(* IEC 61131-3 sources: CodesysTest/alpha/export (part 2) *)

(* ---- ElectricPressureBarFB.st ---- *)
FUNCTION_BLOCK ElectricPressureBarFB IMPLEMENTS IComponentStatus
VAR_INPUT
    enable : BOOL;
END_VAR
VAR_IN_OUT

END_VAR
VAR_OUTPUT
END_VAR
VAR
    electricPressureBarMotor : FB_FestoMotor();
    delay: TON := (PT := T#1S);
    state : PRESSURE_BAR_STATES;
    enableElectricPressureBarONS : R_TRIG();

    _mode : DEVICE_MODES;    // Auto-SemiAuto-Manual
    _ready : BOOL;            // Ready to be controlled
    _amOpenJaw : BOOL;    // Auto Mode Open Jaw Command
    _amCloseJaw : BOOL;     // Auto Mode Close Jaw Command
END_VAR

//    Function Block: ElectricPressureBarFB
//    Description: This function block is the state machine for the electric pressure bar
//
//    Created by: Ben Hess
//    Created Date: Monday, April 16, 2018

electricPressureBarMotor(deviceType := FML.CMMP_AS,
                                        isFPCActive := TRUE,
                                        ptrReadFHPPRegister := ADR(%IW145),
                                        ptrReadFPCRegister := ADR(%IW149),
                                        ptrWriteFHPPRegister := ADR(%QW82),
                                        ptrWriteFPCRegister := ADR(%QW86));
electricPressureBarMotor.Execute();

delay();

//Report as ready if mode is auto and we're not faulted
_ready := (_mode = DEVICE_MODES.Auto) AND NOT (state = PRESSURE_BAR_STATES.Fault);

enableElectricPressureBarONS(CLK := enable);
IF enableElectricPressureBarONS.Q THEN
    state := PRESSURE_BAR_STATES.Idle;
END_IF

IF NOT enable THEN
        state := PRESSURE_BAR_STATES.Fault;
END_IF

CASE state OF
    PRESSURE_BAR_STATES.Idle:        IF enable AND _mode = DEVICE_MODES.SemiAuto OR (_mode = DEVICE_MODES.Auto AND _amCloseJaw) THEN
                                        state := PRESSURE_BAR_STATES.CloseJaw;
                                        _amCloseJaw := FALSE;
                                    END_IF

    PRESSURE_BAR_STATES.OpenJaw:    electricPressureBarMotor.ExecuteStoredProgram(1);
                                    IF electricPressureBarMotor.CommandAcknowledged THEN
                                        state := PRESSURE_BAR_STATES.OpeningJaw;
                                        Globals.electricPressureBarCount := Globals.electricPressureBarCount + 1;
                                    END_IF

    PRESSURE_BAR_STATES.OpeningJaw:
                                    IF electricPressureBarMotor.ActiveStoredProgramNumber = 1 AND electricPressureBarMotor.InPosition THEN
                                        state := PRESSURE_BAR_STATES.JawOpened;
                                    END_IF

    PRESSURE_BAR_STATES.JawOpened:     IF _mode = DEVICE_MODES.SemiAuto THEN
                                        delay.IN := TRUE;
                                        IF delay.Q THEN
                                            state := PRESSURE_BAR_STATES.CloseJaw;
                                            delay.IN := FALSE;
                                        END_IF
                                    ELSIF _mode = DEVICE_MODES.Auto AND _amCloseJaw THEN
                                        state := PRESSURE_BAR_STATES.CloseJaw;
                                        _amCloseJaw := FALSE;
                                    END_IF

    PRESSURE_BAR_STATES.CloseJaw:    electricPressureBarMotor.ExecuteStoredProgram(2);
                                    IF electricPressureBarMotor.CommandAcknowledged THEN
                                        state := PRESSURE_BAR_STATES.ClosingJaw;
                                        Globals.electricPressureBarCount := Globals.electricPressureBarCount + 1;
                                    END_IF

    PRESSURE_BAR_STATES.ClosingJaw:    IF electricPressureBarMotor.ActiveStoredProgramNumber = 2 AND electricPressureBarMotor.InPosition THEN
                                        state := PRESSURE_BAR_STATES.JawClosed;
                                    END_IF

    PRESSURE_BAR_STATES.JawClosed:    IF _mode = DEVICE_MODES.SemiAuto THEN
                                        delay.IN := TRUE;
                                        IF delay.Q THEN
                                            state := PRESSURE_BAR_STATES.OpenJaw;
                                            delay.IN := FALSE;
                                        END_IF
                                    ELSIF _mode = DEVICE_MODES.Auto AND _amOpenJaw THEN
                                        state := PRESSURE_BAR_STATES.OpenJaw;
                                        _amOpenJaw := FALSE;
                                    END_IF

    PRESSURE_BAR_STATES.Fault:        ClearCommands();

END_CASE

METHOD AutoCloseJaw
VAR_INPUT
END_VAR

_amCloseJaw := TRUE;

METHOD AutoOpenJaw
VAR_INPUT
END_VAR

_amOpenJaw := TRUE;

PROPERTY Mode : DEVICE_MODES

PROPERTY Ready : BOOL

METHOD PRIVATE ClearCommands
VAR_INPUT
END_VAR

_amCloseJaw := FALSE;
_amOpenJaw := FALSE;

(* ---- FB_AppliedMotionBagDeliveryMotor.st ---- *)
FUNCTION_BLOCK FB_AppliedMotionBagDeliveryMotor EXTENDS FB_AppliedMotionStepServoTCP
VAR_INPUT
END_VAR
VAR_OUTPUT
END_VAR
VAR
    sendParameters : FB_SendUserRegistersAppliedMotionTCP();
    sendBagMoveCommand : FB_SendBagMoveAppliedMotionTCP();
END_VAR

sendMoveCommand(Slave := slave);
sendBagMoveCommand(Slave := slave);
sendOpcodeCommand(Slave := slave);
sendParameters(Slave := slave);

commandSuccessful S= ((sendMoveCommand.xDone OR sendOpcodeCommand.xDone OR sendBagMoveCommand.xDone) AND NOT status.inPosition) OR sendParameters.xDone;

METHOD MoveDistance
VAR_INPUT
    distance : REAL;        //Distance to move in inches
    acceleration : INT;        //Acceleration in RPM/sec
    deceleration : INT;        //Deceleration in RPM/sec
    velocity : INT;            //Velocity in .25RPM
END_VAR
distanceToMoveInSteps.rawValue := REAL_TO_DINT((distance) * stepsPerInchSetpoint);
IF reversePolarity THEN
    distanceToMoveInSteps.rawValue := distanceToMoveInSteps.rawValue * -1;
END_IF
commandSuccessful := FALSE;
ModbusLongHandler.Unpack(distanceToMoveInSteps);
sendBagMoveCommand.acceleration := acceleration;
sendBagMoveCommand.deceleration := deceleration;
sendBagMoveCommand.velocity := velocity;
sendBagMoveCommand.distanceHighWord := distanceToMoveInSteps.highWord;
sendBagMoveCommand.distanceLowWord := distanceToMoveInSteps.lowWord;
sendBagMoveCommand.opcode := STEP_SERVO_OPCODES.QUEUE_LOAD_AND_EXECUTE;
sendBagMoveCommand.programToRun := 1;
sendBagMoveCommand.Execute();

METHOD SendParameters
VAR_INPUT
    reverseSpeed : DINT;

END_VAR

METHOD MoveDistanceFinal
VAR_INPUT
    distance : REAL;        //Distance to move in inches
    acceleration : INT;        //Acceleration in RPM/sec
    deceleration : INT;        //Deceleration in RPM/sec
    velocity : INT;            //Velocity in .25RPM
END_VAR

distanceToMoveInSteps.rawValue := REAL_TO_DINT((distance) * stepsPerInchSetpoint);
IF reversePolarity THEN
    distanceToMoveInSteps.rawValue := distanceToMoveInSteps.rawValue * -1;
END_IF
commandSuccessful := FALSE;
ModbusLongHandler.Unpack(distanceToMoveInSteps);
sendBagMoveCommand.acceleration := acceleration;
sendBagMoveCommand.deceleration := deceleration;
sendBagMoveCommand.velocity := velocity;
sendBagMoveCommand.distanceHighWord := distanceToMoveInSteps.highWord;
sendBagMoveCommand.distanceLowWord := distanceToMoveInSteps.lowWord;
sendBagMoveCommand.opcode := STEP_SERVO_OPCODES.QUEUE_LOAD_AND_EXECUTE;
sendBagMoveCommand.programToRun := 2;
sendBagMoveCommand.Execute();

METHOD StopViaProgram

// Load program segment 12 into buffer and execute.  This program contains nothing but a SM command.
// We must do it this way because the normal "stop command" opcode we have access to over modbus
// also kills the program buffer which is bad.
commandSuccessful := FALSE;
SendOpcodeCommand.opcode := STEP_SERVO_OPCODES.QUEUE_LOAD_AND_EXECUTE;
SendOpcodeCommand.Parameter1 := INT_TO_WORD(12);    //program 12 is just a SM command
SendOpcodeCommand.Execute();

(* ---- FB_AppliedMotionBagDeliveryMotor_1.st ---- *)
FUNCTION_BLOCK FB_AppliedMotionBagDeliveryMotor_1 EXTENDS FB_AppliedMotionStepServoEIPBase
VAR_INPUT
END_VAR
VAR_OUTPUT
END_VAR
VAR
	_moveDistance : BOOL;
	_moveDistanceONS : R_TRIG;
	_moveFinal : BOOL;
	_moveFinalONS : R_TRIG;
	_moveDone : BOOL;
	waitForMove : TON := (PT := T#30MS);
	manualFinalMovePB : BOOL;
	movedFinal : BOOL;
	moveDistanceState : AMP_EIP_MOVE_INITIAL_STATES;
	moveDistanceFinalState : AMP_EIP_MOVE_INITIAL_STATES;
END_VAR

METHOD Execute
VAR_INPUT
END_VAR

SUPER^.Execute();
waitForMove();
_moveDistanceONS(CLK := _moveDistance);
_moveFinalONS(CLK := _moveFinal);

CASE moveDistanceState OF
	AMP_EIP_MOVE_INITIAL_STATES.Idle :
															IF _moveDistance THEN
																moveDistanceState := AMP_EIP_MOVE_INITIAL_STATES.SetOutputOff;
															END_IF

	AMP_EIP_MOVE_INITIAL_STATES.SetOutputOff :					sclCommand := 16#534F; //Output off
															parameter1 := 16#48B2;
															commands.SendHostCommand := TRUE;
															IF commandSuccessful THEN
																commandSuccessful := FALSE;
																moveDistanceState := AMP_EIP_MOVE_INITIAL_STATES.WaitAfterSettingOutputOff;
															END_IF

	AMP_EIP_MOVE_INITIAL_STATES.WaitAfterSettingOutputOff :
															IF commandSuccessful THEN
																moveDistanceState := AMP_EIP_MOVE_INITIAL_STATES.MoveMotor;
															END_IF

	AMP_EIP_MOVE_INITIAL_STATES.MoveMotor: 					commandSuccessful := FALSE;
															sclCommand := 16#0;
															parameter1 := 16#0;
															commands.FeedToLength := TRUE;
															_moveDistance := FALSE;
															moveDistanceState := AMP_EIP_MOVE_INITIAL_STATES.WaitAfterMovingMotor;

	AMP_EIP_MOVE_INITIAL_STATES.WaitAfterMovingMotor: 		IF commandSuccessful THEN
																_moveDone := TRUE;
																moveDistanceState := AMP_EIP_MOVE_INITIAL_STATES.Idle;
															END_IF
END_CASE

CASE moveDistanceFinalState OF
	AMP_EIP_MOVE_INITIAL_STATES.Idle :						IF _moveFinal THEN
																moveDistanceFinalState := AMP_EIP_MOVE_INITIAL_STATES.SetOutputOff;
															END_IF

	AMP_EIP_MOVE_INITIAL_STATES.SetOutputOff :					sclCommand := 16#534F; //Output off
															parameter1 := 16#48B2;
															commands.SendHostCommand := TRUE;
															IF commandSuccessful THEN
																commandSuccessful := FALSE;
																moveDistanceFinalState := AMP_EIP_MOVE_INITIAL_STATES.WaitAfterSettingOutputOff;
															END_IF

	AMP_EIP_MOVE_INITIAL_STATES.WaitAfterSettingOutputOff :
															IF commandSuccessful THEN
																moveDistanceFinalState := AMP_EIP_MOVE_INITIAL_STATES.MoveMotor;
															END_IF

	AMP_EIP_MOVE_INITIAL_STATES.MoveMotor: 					sclCommand := 16#0;
															parameter1 := 16#0;
															commandSuccessful := FALSE;
															commands.FeedToLength := TRUE;
															moveDistanceFinalState := AMP_EIP_MOVE_INITIAL_STATES.WaitAfterMovingMotor;

	AMP_EIP_MOVE_INITIAL_STATES.WaitAfterMovingMotor: 		IF commandSuccessful AND InPosition THEN
																moveDistanceFinalState := AMP_EIP_MOVE_INITIAL_STATES.SetOutputOn;
															END_IF

	AMP_EIP_MOVE_INITIAL_STATES.SetOutputOn :					sclCommand := 16#534F; // Output on
															parameter1 := 16#4CB2;

															commandSuccessful := FALSE;
															commands.SendHostCommand := TRUE;
															_moveFinal := FALSE;
															moveDistanceFinalState := AMP_EIP_MOVE_INITIAL_STATES.WaitAfterSettingOutputOn;

	AMP_EIP_MOVE_INITIAL_STATES.WaitAfterSettingOutputOn :
															IF commandSuccessful THEN
																_moveDone := TRUE;
																moveDistanceFinalState := AMP_EIP_MOVE_INITIAL_STATES.Idle;
															END_IF

END_CASE
(*
IF _moveFinal THEN
	IF NOT movedFinal AND commandSuccessful THEN
		commandSuccessful := FALSE;
		commands.FeedToLength := TRUE;
		waitForMove.IN := TRUE;
		movedFinal := TRUE;
	END_IF

	IF commandSuccessful AND waitForMove.Q AND InPosition THEN
		sclCommand := 16#534F;
		parameter1 := 16#4CB2;
		commands.SendHostCommand := TRUE;
		_moveFinal := FALSE;
		waitForMove.IN := FALSE;
		movedFinal := FALSE;
	END_IF
END_IF
*)
IF manualFinalMovePB THEN
    MoveDistanceFinal(distance := distanceSetpointInches, acceleration := pointToPointAccelSetpoint, deceleration := pointToPointDecelSetpoint, velocity := velocitySetpoint);
    manualFinalMovePB := FALSE;
END_IF

PROPERTY CommandAcknowledged : BOOL

METHOD SetRearMotorToTorqueMode
VAR_INPUT
END_VAR

sclCommand := 16#534F; // Output on
parameter1 := 16#4CB2;

commandSuccessful := FALSE;
commands.SendHostCommand := TRUE;

METHOD SetRearMotorToEncoderFollowing
VAR_INPUT
END_VAR

METHOD StopViaProgram

// Load program segment 12 into buffer and execute.  This program contains nothing but a SM command.
// We must do it this way because the normal "stop command" opcode we have access to over modbus
// also kills the program buffer which is bad.
SUPER^.Stop();

METHOD MoveDistanceFinal
VAR_INPUT
    distance : REAL;        //Distance to move in inches
    acceleration : INT;        //Acceleration in RPM/sec
    deceleration : INT;        //Deceleration in RPM/sec
    velocity : INT;            //Velocity in .25RPM
END_VAR

commandSuccessful := FALSE;
_moveDone := FALSE;
moveDistanceFinalState := AMP_EIP_MOVE_INITIAL_STATES.Idle;
distanceToMoveInSteps := REAL_TO_DINT((distance) * stepsPerInchSetpoint);
IF reversePolarity THEN
    distanceToMoveInSteps := distanceToMoveInSteps * -1;
END_IF

pointToPointAccelSetpoint := acceleration;
pointToPointDecelSetpoint := deceleration;
velocitySetpoint := velocity;

currentLimit := defaultCurrentSetpoint;
_moveFinal := TRUE;
//SUPER^.ExecuteStoredProgram(2);

METHOD MoveDistance
VAR_INPUT
    distance : REAL;        //Distance to move in inches
    acceleration : INT;        //Acceleration in RPM/sec
    deceleration : INT;        //Deceleration in RPM/sec
    velocity : INT;            //Velocity in .25RPM
END_VAR
commandSuccessful := FALSE;
_moveDone := FALSE;
moveDistanceState := AMP_EIP_MOVE_INITIAL_STATES.Idle;
distanceToMoveInSteps := REAL_TO_DINT((distance) * stepsPerInchSetpoint);

IF reversePolarity THEN
    distanceToMoveInSteps := distanceToMoveInSteps * -1;
END_IF

pointToPointAccelSetpoint := acceleration;
pointToPointDecelSetpoint := deceleration;
velocitySetpoint := velocity;

currentLimit := defaultCurrentSetpoint;
_moveDistance := TRUE;

//commands.feedToLength := TRUE;
//SUPER^.ExecuteStoredProgram(1);

(* ---- FB_AppliedMotionBagDeliveryMotorNoFollowing.st ---- *)
FUNCTION_BLOCK FB_AppliedMotionBagDeliveryMotorNoFollowing EXTENDS FB_AppliedMotionStepServoEIPBase
VAR_INPUT
END_VAR
VAR_OUTPUT
END_VAR
VAR
	_moveDistance : BOOL;
	_moveDistanceONS : R_TRIG;
	_moveFinal : BOOL;
	_moveFinalONS : R_TRIG;
	_moveDone : BOOL;
	waitForMove : TON := (PT := T#30MS);
	manualFinalMovePB : BOOL;
	movedFinal : BOOL;
	moveDistanceState : AMP_EIP_MOVE_INITIAL_STATES;
	moveDistanceFinalState : AMP_EIP_MOVE_INITIAL_STATES;
END_VAR

METHOD Execute
VAR_INPUT
END_VAR

SUPER^.Execute();
waitForMove();
_moveDistanceONS(CLK := _moveDistance);
_moveFinalONS(CLK := _moveFinal);

CASE moveDistanceState OF
	AMP_EIP_MOVE_INITIAL_STATES.Idle :
															IF _moveDistance THEN
																moveDistanceState := AMP_EIP_MOVE_INITIAL_STATES.SetOutputOff;
															END_IF

	AMP_EIP_MOVE_INITIAL_STATES.SetOutputOff :					sclCommand := 16#534F; //Output off
															parameter1 := 16#48B2;
															commands.SendHostCommand := TRUE;
															IF commandSuccessful THEN
																commandSuccessful := FALSE;
																moveDistanceState := AMP_EIP_MOVE_INITIAL_STATES.WaitAfterSettingOutputOff;
															END_IF

	AMP_EIP_MOVE_INITIAL_STATES.WaitAfterSettingOutputOff :
															IF commandSuccessful THEN
																moveDistanceState := AMP_EIP_MOVE_INITIAL_STATES.MoveMotor;
															END_IF

	AMP_EIP_MOVE_INITIAL_STATES.MoveMotor: 					commandSuccessful := FALSE;
															sclCommand := 16#0;
															parameter1 := 16#0;
															commands.FeedToLength := TRUE;
															_moveDistance := FALSE;
															moveDistanceState := AMP_EIP_MOVE_INITIAL_STATES.WaitAfterMovingMotor;

	AMP_EIP_MOVE_INITIAL_STATES.WaitAfterMovingMotor: 		IF commandSuccessful THEN
																_moveDone := TRUE;
																moveDistanceState := AMP_EIP_MOVE_INITIAL_STATES.Idle;
															END_IF
END_CASE

CASE moveDistanceFinalState OF
	AMP_EIP_MOVE_INITIAL_STATES.Idle :						IF _moveFinal THEN
																moveDistanceFinalState := AMP_EIP_MOVE_INITIAL_STATES.MoveMotor;
															END_IF

	AMP_EIP_MOVE_INITIAL_STATES.MoveMotor: 					sclCommand := 16#0;
															parameter1 := 16#0;
															commandSuccessful := FALSE;
															commands.FeedToLength := TRUE;
															moveDistanceFinalState := AMP_EIP_MOVE_INITIAL_STATES.WaitAfterMovingMotor;

	AMP_EIP_MOVE_INITIAL_STATES.WaitAfterMovingMotor: 		IF commandSuccessful AND InPosition THEN
																moveDistanceFinalState := AMP_EIP_MOVE_INITIAL_STATES.SetOutputOff;
															END_IF

	AMP_EIP_MOVE_INITIAL_STATES.SetOutputOff :					sclCommand := 16#534F; // Output on
															parameter1 := 16#4CB2;

															commandSuccessful := FALSE;
															commands.SendHostCommand := TRUE;
															_moveFinal := FALSE;
															moveDistanceFinalState := AMP_EIP_MOVE_INITIAL_STATES.WaitAfterSettingOutputOff;

	AMP_EIP_MOVE_INITIAL_STATES.WaitAfterSettingOutputOff :
															IF commandSuccessful THEN
																_moveDone := TRUE;
																moveDistanceFinalState := AMP_EIP_MOVE_INITIAL_STATES.Idle;
															END_IF

END_CASE
(*
IF _moveFinal THEN
	IF NOT movedFinal AND commandSuccessful THEN
		commandSuccessful := FALSE;
		commands.FeedToLength := TRUE;
		waitForMove.IN := TRUE;
		movedFinal := TRUE;
	END_IF

	IF commandSuccessful AND waitForMove.Q AND InPosition THEN
		sclCommand := 16#534F;
		parameter1 := 16#4CB2;
		commands.SendHostCommand := TRUE;
		_moveFinal := FALSE;
		waitForMove.IN := FALSE;
		movedFinal := FALSE;
	END_IF
END_IF
*)
IF manualFinalMovePB THEN
    MoveDistanceFinal(distance := distanceSetpointInches, acceleration := pointToPointAccelSetpoint, deceleration := pointToPointDecelSetpoint, velocity := velocitySetpoint);
    manualFinalMovePB := FALSE;
END_IF

PROPERTY CommandAcknowledged : BOOL

METHOD SetRearMotorToTorqueMode
VAR_INPUT
END_VAR

METHOD SetRearMotorToEncoderFollowing
VAR_INPUT
END_VAR

METHOD StopViaProgram

// Load program segment 12 into buffer and execute.  This program contains nothing but a SM command.
// We must do it this way because the normal "stop command" opcode we have access to over modbus
// also kills the program buffer which is bad.
SUPER^.Stop();

METHOD MoveDistanceFinal
VAR_INPUT
    distance : REAL;        //Distance to move in inches
    acceleration : INT;        //Acceleration in RPM/sec
    deceleration : INT;        //Deceleration in RPM/sec
    velocity : INT;            //Velocity in .25RPM
END_VAR

commandSuccessful := FALSE;
_moveDone := FALSE;
moveDistanceFinalState := AMP_EIP_MOVE_INITIAL_STATES.Idle;
distanceToMoveInSteps := REAL_TO_DINT((distance) * stepsPerInchSetpoint);
IF reversePolarity THEN
    distanceToMoveInSteps := distanceToMoveInSteps * -1;
END_IF

pointToPointAccelSetpoint := acceleration;
pointToPointDecelSetpoint := deceleration;
velocitySetpoint := velocity;

currentLimit := defaultCurrentSetpoint;
_moveFinal := TRUE;
//SUPER^.ExecuteStoredProgram(2);

METHOD MoveDistance
VAR_INPUT
    distance : REAL;        //Distance to move in inches
    acceleration : INT;        //Acceleration in RPM/sec
    deceleration : INT;        //Deceleration in RPM/sec
    velocity : INT;            //Velocity in .25RPM
END_VAR
commandSuccessful := FALSE;
_moveDone := FALSE;
moveDistanceState := AMP_EIP_MOVE_INITIAL_STATES.Idle;
distanceToMoveInSteps := REAL_TO_DINT((distance) * stepsPerInchSetpoint);

IF reversePolarity THEN
    distanceToMoveInSteps := distanceToMoveInSteps * -1;
END_IF

pointToPointAccelSetpoint := acceleration;
pointToPointDecelSetpoint := deceleration;
velocitySetpoint := velocity;

currentLimit := defaultCurrentSetpoint;
_moveDistance := TRUE;

//commands.feedToLength := TRUE;
//SUPER^.ExecuteStoredProgram(1);

(* ---- FB_AppliedMotionStepServoEIPBase.st ---- *)
FUNCTION_BLOCK FB_AppliedMotionStepServoEIPBase IMPLEMENTS IPositionableMotor, IStoredProgramMotor
VAR_INPUT
    ptrEIPInputs : POINTER TO ARRAY[0..13] OF  DINT;
    ptrEIPOutputs : POINTER TO ARRAY[0..15] OF DINT;
    faultHandler : REFERENCE TO FB_FaultHandler;
	commFail : BOOL;
    stepsPerInchSetpoint : INT;             //Steps per inch setpoint
    reversePolarity : BOOL;                 //0 = Normal, 1 = reversed polarity for display
    jogAccelSetpoint : INT;        //Point-to-Point Acceleration (AC) Setpoint
    jogDecelSetpoint : INT;        //Point-to-Point Deceleration (DE) Setpoint
    jogVelocitySetpoint : INT;                //Velocity (VE) Setpoint
    pointToPointAccelSetpoint : INT;        //Point-to-Point Acceleration (AC) Setpoint
    pointToPointDecelSetpoint : INT;        //Point-to-Point Deceleration (DE) Setpoint
    velocitySetpoint : INT;                //Velocity (VE) Setpoint
	defaultCurrentSetpoint : DINT;
	sclCommand : DINT;						// SCL Command from
	parameter1 : DINT;						// Data/SCL parameter 1
	parameter2 : DINT;						// Data/SCL parameter 2
    distanceSetpointInches : REAL;        //Distance setpoint in inches Setpoint
    moveDistanceManualPB : BOOL;            //Move distance pushbutton
    movePositionManualPB : BOOL;            //Move position pushbutton
	isHomable : BOOL;
END_VAR
VAR_IN_OUT
    //slave : IoDrvModbusTCP.ModbusTCPSlave;                    //Slave ModbusTCP Object
END_VAR
VAR
    absolutePositionSteps : DINT; //Immediate Absolute Position in steps
    distanceToMoveInSteps : DINT;        //Distance Setpoint to Drive
    stepServoStatusRaw : INT; //Raw step servo status over modbus
	stepServoAlarmCodeRaw : INT; // Ras Step Servo alarm code word
	currentLimit : DINT;
    commands : FB_StepServoCommands();
    commandSuccessful : BOOL;    //Modbus Command was successful
    commandSuccessfulONS : R_TRIG;    //Modbus Command was successful
    commandSentONS : R_TRIG;    //Modbus Command was successful
    homeRequiredIndication : BOOL; //Home required indication.
    driveInputs : ARRAY[0..13] OF DINT;        // Inputs from drive over EIP
    driveOutputs : ARRAY[0..15] OF DINT;    // Outputs to drive over EIP
    interfaceToPass : IFault;
    faultListRegisterSuccess : BOOL;        // Registering in fault list successful
    _faulted : BOOL;                    // Motor Faulted
	_reset : BOOL;			//Reset Motor
	_homeNow : BOOL;
	homingOSF : F_TRIG;

	IECReferenceGood : BOOL;
END_VAR
VAR_OUTPUT
    absolutePositonInches : REAL; //Immediate Absolute Positon in inches
    velocity : INT;    //Velocity (VE) Input from Drive
    status : StepServoStatusFB; //Status of servo
	alarms : FB_StepServoAlarms; // Alarms from Drive
    QSegmentRunning : INT; //Current Q program running from Drive
	faults : StepServoFaultsType;
END_VAR

IF NOT faultListRegisterSuccess THEN
    faultListRegisterSuccess := RegisterWithFaultHandler();
END_IF

{attribute 'monitoring' := 'variable'}
PROPERTY HomeRequired : BOOL

{attribute 'monitoring' := 'variable'}
PROPERTY InPosition : BOOL

//{warning 'add method implementation '}
METHOD Stop

commandSuccessful := FALSE;
commands.StopNormal := TRUE;

METHOD RegisterWithFaultHandler : BOOL

// If faulthandler hasn't been initialized yet then do nothing.

(*
IF NOT __ISVALIDREF(faultHandler) THEN
     RETURN;
END_IF

interfaceToPass := THIS^;
faultHandler.registerFaultSource(interfaceToPass);
RegisterWithFaultHandler := TRUE;
*)

{attribute 'monitoring' := 'variable'}
PROPERTY Faulted : BOOL

{attribute 'monitoring' := 'variable'}
PROPERTY Homing : BOOL

METHOD Execute
VAR_INPUT
END_VAR

//    Function Block: AppliedMotionStepServo
//    Description: This block provides an abstraction for a Ethernet I/P Applied Motion Step Servo
//    Created by: Ben Hess
//    Created Date: May 11th, 2018

// Use pointers for EIP memory register locations
driveInputs := ptrEIPInputs^;
// Step servo command bits handler
commands();
ptrEIPOutputs^ := driveOutputs;
alarms(alarmCode := stepServoAlarmCodeRaw, faults := faults);

IF currentLimit = 0 THEN
	currentLimit := defaultCurrentSetpoint;
END_IF
//Map raw EIP Registers to parameters
absolutePositionSteps := driveInputs[6];
velocity := DINT_TO_INT(driveInputs[8]);
stepServoStatusRaw := DINT_TO_INT(driveInputs[0]);

driveOutputs[4] := velocitySetpoint;
driveOutputs[5] := pointToPointAccelSetpoint;
driveOutputs[6] := pointToPointDecelSetpoint;
driveOutputs[7] := distanceToMoveInSteps;
driveOutputs[8] := currentLimit;
driveOutputs[9] := sclCommand;
driveOutputs[10] := parameter1;
driveOutputs[11] := parameter2;
driveOutputs[12] := currentLimit;
driveOutputs[13] := currentLimit + 1;
driveOutputs[0] := commands.commandWord;

//Convert Distance setpoint to steps.  Reverse polarity for display purposes if needed.

absolutePositonInches := (DINT_TO_REAL(absolutePositionSteps) / INT_TO_REAL(stepsPerInchSetpoint));

//Homing required from motor - for now just if there was an initialization seen.
homeRequiredIndication S= status.initializing OR Globals.firstScan OR _faulted OR driveInputs[11].0;

homingOSF(CLK := status.homing);
IF NOT driveInputs[11].0 THEN
	homeRequiredIndication := FALSE;
END_IF

commandSentONS(CLK := commands.commandSent);

IF commandSentONS.Q THEN
	commandSuccessful := TRUE;
END_IF

commandSuccessfulONS(CLK := commandSuccessful);
IF commandSuccessfulONS.Q THEN
	//parameter1 := 0;
	//velocitySetpoint := 0;
	//pointToPointAccelSetpoint := 0;
	//pointToPointDecelSetpoint := 0;
	//distanceToMoveInSteps := 0;
END_IF

IF _reset AND (status.driveFaulted OR status.alarmPresent) THEN
	commands.alarmReset := TRUE;
	_reset := FALSE;
END_IF

IF reversePolarity THEN
    absolutePositonInches := absolutePositonInches * -1;
END_IF

//Get Servo Status and unpack
status(statusCode := StepServoStatusRaw);

//Bit-packing for LONG types over Modbus

_faulted := status.driveFaulted OR status.alarmPresent OR commFail;

//Manual moves for motor
IF moveDistanceManualPB THEN
    MoveDistance(distance := distanceSetpointInches, acceleration := pointToPointAccelSetpoint, deceleration := pointToPointDecelSetpoint, velocity := velocitySetpoint);
    moveDistanceManualPB := FALSE;
END_IF

IF movePositionManualPB THEN
    MoveToPosition(position := distanceSetpointInches, acceleration := pointToPointAccelSetpoint, deceleration := pointToPointDecelSetpoint, velocity := velocitySetpoint);
    movePositionManualPB := FALSE;
END_IF

faults.commFail.faultTrigger := commFail AND Globals.machinePowerOK;
faults.notHomed.faultTrigger := homeRequiredIndication AND isHomable;

METHOD MoveDistance
VAR_INPUT
    (*Distance to move in inches*)
    distance    : REAL;
    (*Acceleration in RPM/sec*)
    acceleration    : INT;
    (*Deceleration in RPM/sec*)
    deceleration    : INT;
    (*Velocity in .25RPM*)
    velocity    : INT;
END_VAR

//This method preps the data to send to the drive and triggers the send.
//Set distance and unpack to prep data to send to motor

commandSuccessful := FALSE;

distanceToMoveInSteps := REAL_TO_DINT((distance) * stepsPerInchSetpoint);
IF reversePolarity THEN
    distanceToMoveInSteps := distanceToMoveInSteps * -1;
END_IF

pointToPointAccelSetpoint := acceleration;
pointToPointDecelSetpoint := deceleration;
velocitySetpoint := velocity;
currentLimit := defaultCurrentSetpoint;

commands.feedToLength := TRUE;

METHOD HomeNow
commandSuccessful := FALSE;
parameter1 := 1;
pointToPointAccelSetpoint := 1000;
pointToPointDecelSetpoint := 1000;
velocitySetpoint := 2500;
distanceToMoveInSteps := 0;
commands.sendQAndExecute := TRUE;

//homeRequiredIndication := FALSE;

{attribute 'monitoring' := 'variable'}
PROPERTY CurrentPosition : REAL  //Current motor position in Inches

METHOD ExecuteStoredProgram
VAR_INPUT
    (*Program number to execute*)
    programNumber    : INT;
END_VAR

parameter1 := programNumber;
commands.SendQAndExecute := TRUE;

{attribute 'monitoring' := 'variable'}
PROPERTY Moving : BOOL

{attribute 'monitoring' := 'variable'}
PROPERTY ActiveStoredProgramNumber : INT

METHOD MoveDistanceTorque
VAR_INPUT
	(*Distance to move in inches*)
    distance    : REAL;
    (*Acceleration in RPM/sec*)
    acceleration    : INT;
    (*Deceleration in RPM/sec*)
    deceleration    : INT;
    (*Velocity in .25RPM*)
    velocity    : INT;
	(*Current in .01A*)
	current : DINT;
END_VAR

//This method preps the data to send to the drive and triggers the send.
//Set distance and unpack to prep data to send to motor

commandSuccessful := FALSE;

distanceToMoveInSteps := REAL_TO_DINT((distance) * stepsPerInchSetpoint);
IF reversePolarity THEN
    distanceToMoveInSteps := distanceToMoveInSteps * -1;
END_IF

pointToPointAccelSetpoint := acceleration;
pointToPointDecelSetpoint := deceleration;
velocitySetpoint := velocity;
currentLimit := current;

commands.feedToLength := TRUE;

METHOD Reset : BOOL
VAR_INPUT
END_VAR

IF Faulted THEN
	_reset := TRUE;
	commands.AlarmReset := TRUE;
END_IF
commands.Enable := TRUE;

{attribute 'monitoring' := 'variable'}
PROPERTY CommandAcknowledged : BOOL

(* ---- FB_AppliedMotionStepServoEIPBaseQX.st ---- *)
FUNCTION_BLOCK FB_AppliedMotionStepServoEIPBaseQX IMPLEMENTS IPositionableMotor, IStoredProgramMotor
VAR_INPUT
    ptrEIPInputs : POINTER TO ARRAY[0..13] OF  DINT;
    ptrEIPOutputs : POINTER TO ARRAY[0..15] OF DINT;
    faultHandler : REFERENCE TO FB_FaultHandler;
	commFail : BOOL;
    stepsPerInchSetpoint : INT;             //Steps per inch setpoint
    reversePolarity : BOOL;                 //0 = Normal, 1 = reversed polarity for display
    jogAccelSetpoint : INT;        //Point-to-Point Acceleration (AC) Setpoint
    jogDecelSetpoint : INT;        //Point-to-Point Deceleration (DE) Setpoint
    jogVelocitySetpoint : INT;                //Velocity (VE) Setpoint
    pointToPointAccelSetpoint : INT;        //Point-to-Point Acceleration (AC) Setpoint
    pointToPointDecelSetpoint : INT;        //Point-to-Point Deceleration (DE) Setpoint
    velocitySetpoint : INT;                //Velocity (VE) Setpoint
	defaultCurrentSetpoint : DINT;
	sclCommand : DINT;						// SCL Command from
	parameter1 : DINT;						// Data/SCL parameter 1
	parameter2 : DINT;						// Data/SCL parameter 2
    distanceSetpointInches : REAL;        //Distance setpoint in inches Setpoint
    moveDistanceManualPB : BOOL;            //Move distance pushbutton
    movePositionManualPB : BOOL;            //Move position pushbutton
	isHomable : BOOL;
END_VAR
VAR_IN_OUT
    //slave : IoDrvModbusTCP.ModbusTCPSlave;                    //Slave ModbusTCP Object
END_VAR
VAR
    absolutePositionSteps : DINT; //Immediate Absolute Position in steps
    distanceToMoveInSteps : DINT;        //Distance Setpoint to Drive
    stepServoStatusRaw : INT; //Raw step servo status over modbus
	stepServoAlarmCodeRaw : INT; // Ras Step Servo alarm code word
	currentLimit : DINT;
    commands : FB_StepServoCommands();
    commandSuccessful : BOOL;    //Modbus Command was successful
    commandSuccessfulONS : R_TRIG;    //Modbus Command was successful
    commandSentONS : R_TRIG;    //Modbus Command was successful
    homeRequiredIndication : BOOL; //Home required indication.
    driveInputs : ARRAY[0..13] OF DINT;        // Inputs from drive over EIP
    driveOutputs : ARRAY[0..15] OF DINT;    // Outputs to drive over EIP
    interfaceToPass : IFault;
    faultListRegisterSuccess : BOOL;        // Registering in fault list successful
    _faulted : BOOL;                    // Motor Faulted
	_reset : BOOL;			//Reset Motor
	_homeNow : BOOL;
	homingOSF : F_TRIG;

	IECReferenceGood : BOOL;
END_VAR
VAR_OUTPUT
    absolutePositonInches : REAL; //Immediate Absolute Positon in inches
    velocity : INT;    //Velocity (VE) Input from Drive
    status : StepServoStatusFB; //Status of servo
	alarms : FB_StepServoAlarms; // Alarms from Drive
    QSegmentRunning : INT; //Current Q program running from Drive
	faults : StepServoFaultsType;
END_VAR

IF NOT faultListRegisterSuccess THEN
    faultListRegisterSuccess := RegisterWithFaultHandler();
END_IF

METHOD Execute
VAR_INPUT
END_VAR

//    Function Block: AppliedMotionStepServo
//    Description: This block provides an abstraction for a Ethernet I/P Applied Motion Step Servo
//    Created by: Ben Hess
//    Created Date: May 11th, 2018

// Use pointers for EIP memory register locations
driveInputs := ptrEIPInputs^;

ptrEIPOutputs^ := driveOutputs;
alarms(alarmCode := stepServoAlarmCodeRaw, faults := faults);

IF currentLimit = 0 THEN
	currentLimit := defaultCurrentSetpoint;
END_IF
//Map raw EIP Registers to parameters
absolutePositionSteps := driveInputs[6];
velocity := DINT_TO_INT(driveInputs[8]);
stepServoStatusRaw := DINT_TO_INT(driveInputs[0]);

driveOutputs[4] := velocitySetpoint;
driveOutputs[5] := pointToPointAccelSetpoint;
driveOutputs[6] := pointToPointDecelSetpoint;
driveOutputs[7] := distanceToMoveInSteps;
driveOutputs[8] := currentLimit;
driveOutputs[9] := sclCommand;
driveOutputs[10] := parameter1;
driveOutputs[11] := parameter2;
driveOutputs[12] := currentLimit;
driveOutputs[13] := currentLimit + 1;
driveOutputs[0] := commands.commandWord;
// Step servo command bits handler
commands();
//Convert Distance setpoint to steps.  Reverse polarity for display purposes if needed.

absolutePositonInches := (DINT_TO_REAL(absolutePositionSteps) / INT_TO_REAL(stepsPerInchSetpoint));

//Homing required from motor - for now just if there was an initialization seen.
homeRequiredIndication S= status.initializing OR Globals.firstScan OR _faulted OR driveInputs[11].0;

homingOSF(CLK := status.homing);
IF NOT driveInputs[11].0 THEN
	homeRequiredIndication := FALSE;
END_IF

commandSentONS(CLK := commands.commandSent);

IF commandSentONS.Q THEN
	commandSuccessful := TRUE;
END_IF

commandSuccessfulONS(CLK := commandSuccessful);
IF commandSuccessfulONS.Q THEN
	//parameter1 := 0;
	//velocitySetpoint := 0;
	//pointToPointAccelSetpoint := 0;
	//pointToPointDecelSetpoint := 0;
	//distanceToMoveInSteps := 0;
END_IF

IF _reset AND (status.driveFaulted OR status.alarmPresent) THEN
	commands.alarmReset := TRUE;
	_reset := FALSE;
END_IF

IF reversePolarity THEN
    absolutePositonInches := absolutePositonInches * -1;
END_IF

//Get Servo Status and unpack
status(statusCode := StepServoStatusRaw);

//Bit-packing for LONG types over Modbus

_faulted := status.driveFaulted OR status.alarmPresent OR commFail;

//Manual moves for motor
IF moveDistanceManualPB THEN
    MoveDistance(distance := distanceSetpointInches, acceleration := pointToPointAccelSetpoint, deceleration := pointToPointDecelSetpoint, velocity := velocitySetpoint);
    moveDistanceManualPB := FALSE;
END_IF

IF movePositionManualPB THEN
    MoveToPosition(position := distanceSetpointInches, acceleration := pointToPointAccelSetpoint, deceleration := pointToPointDecelSetpoint, velocity := velocitySetpoint);
    movePositionManualPB := FALSE;
END_IF

faults.commFail.faultTrigger := commFail AND Globals.machinePowerOK;
faults.notHomed.faultTrigger := homeRequiredIndication AND isHomable;

{attribute 'monitoring' := 'variable'}
PROPERTY CommandAcknowledged : BOOL

METHOD HomeNow
commandSuccessful := FALSE;
parameter1 := 1;
pointToPointAccelSetpoint := 1000;
pointToPointDecelSetpoint := 1000;
velocitySetpoint := 2500;
distanceToMoveInSteps := 0;
commands.sendQAndExecute := TRUE;

//homeRequiredIndication := FALSE;

{attribute 'monitoring' := 'variable'}
PROPERTY Homing : BOOL

{attribute 'monitoring' := 'variable'}
PROPERTY HomeRequired : BOOL

{attribute 'monitoring' := 'variable'}
PROPERTY Moving : BOOL

{attribute 'monitoring' := 'variable'}
PROPERTY ActiveStoredProgramNumber : INT

{attribute 'monitoring' := 'variable'}
PROPERTY InPosition : BOOL

METHOD MoveDistanceTorque
VAR_INPUT
	(*Distance to move in inches*)
    distance    : REAL;
    (*Acceleration in RPM/sec*)
    acceleration    : INT;
    (*Deceleration in RPM/sec*)
    deceleration    : INT;
    (*Velocity in .25RPM*)
    velocity    : INT;
	(*Current in .01A*)
	current : DINT;
END_VAR

//This method preps the data to send to the drive and triggers the send.
//Set distance and unpack to prep data to send to motor

commandSuccessful := FALSE;

distanceToMoveInSteps := REAL_TO_DINT((distance) * stepsPerInchSetpoint);
IF reversePolarity THEN
    distanceToMoveInSteps := distanceToMoveInSteps * -1;
END_IF

pointToPointAccelSetpoint := acceleration;
pointToPointDecelSetpoint := deceleration;
velocitySetpoint := velocity;
currentLimit := current;

parameter1 := 2;
commands.SendQAndExecute := TRUE;

(* This will be called if the machine is faulted*)
METHOD MachineFaulted

{attribute 'monitoring' := 'variable'}
PROPERTY Faulted : BOOL

METHOD MoveToPosition
VAR_INPUT
    (*Position to move to in inches*)
    position    : REAL;
    (*Acceleration in RPM/sec*)
    acceleration    : INT;
    (*Deceleration in RPM/sec*)
    deceleration    : INT;
    (*Velocity in .25RPM*)
    velocity    : INT;
END_VAR

commandSuccessful := FALSE;

distanceToMoveInSteps := REAL_TO_DINT((position) * stepsPerInchSetpoint);
IF reversePolarity THEN
    distanceToMoveInSteps := distanceToMoveInSteps * -1;
END_IF

pointToPointAccelSetpoint := acceleration;
pointToPointDecelSetpoint := deceleration;
velocitySetpoint := velocity;
currentLimit := defaultCurrentSetpoint;

commands.feedToPosition := TRUE;

METHOD MoveToPositionTorque
VAR_INPUT
	(*Position to move to in inches*)
    position    : REAL;
    (*Acceleration in RPM/sec*)
    acceleration    : INT;
    (*Deceleration in RPM/sec*)
    deceleration    : INT;
    (*Velocity in .25RPM*)
    velocity    : INT;
	(*Current in .01A*)
	current : DINT;
END_VAR

commandSuccessful := FALSE;

distanceToMoveInSteps := REAL_TO_DINT((position) * stepsPerInchSetpoint);
IF reversePolarity THEN
    distanceToMoveInSteps := distanceToMoveInSteps * -1;
END_IF

pointToPointAccelSetpoint := acceleration;
pointToPointDecelSetpoint := deceleration;
velocitySetpoint := velocity;
currentLimit := current;

commands.feedToPosition := TRUE;
THIS^.Execute();

//{warning 'add method implementation '}
METHOD Stop

commandSuccessful := FALSE;
commands.StopNormal := TRUE;

METHOD MoveDistance
VAR_INPUT
    (*Distance to move in inches*)
    distance    : REAL;
    (*Acceleration in RPM/sec*)
    acceleration    : INT;
    (*Deceleration in RPM/sec*)
    deceleration    : INT;
    (*Velocity in .25RPM*)
    velocity    : INT;
END_VAR

//This method preps the data to send to the drive and triggers the send.
//Set distance and unpack to prep data to send to motor

commandSuccessful := FALSE;

distanceToMoveInSteps := REAL_TO_DINT((distance) * stepsPerInchSetpoint);
IF reversePolarity THEN
    distanceToMoveInSteps := distanceToMoveInSteps * -1;
END_IF

pointToPointAccelSetpoint := acceleration;
pointToPointDecelSetpoint := deceleration;
velocitySetpoint := velocity;
currentLimit := defaultCurrentSetpoint;

commands.feedToLength := TRUE;

{attribute 'monitoring' := 'variable'}
PROPERTY CurrentPosition : REAL  //Current motor position in Inches

METHOD Reset : BOOL
VAR_INPUT
END_VAR

IF Faulted THEN
	_reset := TRUE;
	commands.AlarmReset := TRUE;
END_IF
commands.Enable := TRUE;

METHOD RegisterWithFaultHandler : BOOL

// If faulthandler hasn't been initialized yet then do nothing.

(*
IF NOT __ISVALIDREF(faultHandler) THEN
     RETURN;
END_IF

interfaceToPass := THIS^;
faultHandler.registerFaultSource(interfaceToPass);
RegisterWithFaultHandler := TRUE;
*)

METHOD ExecuteStoredProgram
VAR_INPUT
    (*Program number to execute*)
    programNumber    : INT;
END_VAR

parameter1 := programNumber;
commands.SendQAndExecute := TRUE;

(* ---- FB_AppliedMotionStepServoEIPPassthrough.st ---- *)
FUNCTION_BLOCK FB_AppliedMotionStepServoEIPPassthrough EXTENDS FB_AppliedMotionStepServoEIPBase
VAR_INPUT
END_VAR
VAR_OUTPUT
END_VAR
VAR
	homingState : JAW_HOMING_STATES;
	homeRequiredONS : R_TRIG;
	timerHomeDelay : TON;
END_VAR

SUPER^();

METHOD Execute
VAR_INPUT
END_VAR

SUPER^.Execute();
timerHomeDelay();
homeRequiredONS(CLK := homeRequiredIndication);

//IF _reset OR homeRequiredONS.Q THEN
IF _reset THEN
	homingState := JAW_HOMING_STATES.Idle;
	_homeNow := FALSE;
	timerHomeDelay.IN := FALSE;
	_reset := FALSE;
END_IF

CASE homingState OF
	JAW_HOMING_STATES.Idle:						IF _homeNow THEN
													IF NOT driveInputs[10].2 THEN
														homingState := JAW_HOMING_STATES.MoveForwardFromSensor;
													ELSE
														homingState := JAW_HOMING_STATES.StartHoming;
													END_IF
													_homeNow := FALSE;
												END_IF

	JAW_HOMING_STATES.MoveForwardFromSensor:	commandSuccessful := FALSE;
												velocitySetpoint := 2583;
												pointToPointAccelSetpoint := 1000;
												pointToPointDecelSetpoint := 1000;
												distanceToMoveInSteps := -4000;
												commands.FeedToLength := TRUE;
												homingState := JAW_HOMING_STATES.MovingForwardFromSensor;

	JAW_HOMING_STATES.MovingForwardFromSensor:	timerHomeDelay.PT := T#200MS;
												timerHomeDelay.IN := TRUE;
												IF timerHomeDelay.Q THEN
													IF (NOT Moving AND InPosition) THEN
														homingState := JAW_HOMING_STATES.StartHoming;
														timerHomeDelay.IN := FALSE;
                                                       END_IF
												END_IF

	JAW_HOMING_STATES.StartHoming:				commandSuccessful := FALSE;
												velocitySetpoint := 2583;
												pointToPointAccelSetpoint := 1000;
												pointToPointDecelSetpoint := 1000;
												distanceToMoveInSteps := 1;
												ExecuteStoredProgram(2);
												homingState := JAW_HOMING_STATES.Homing;

	JAW_HOMING_STATES.Homing:					timerHomeDelay.PT := T#200MS;
												timerHomeDelay.IN := TRUE;
												IF timerHomeDelay.Q THEN
													IF (NOT SUPER^.Homing) THEN
														homingState := JAW_HOMING_STATES.HomeComplete;
														timerHomeDelay.IN := FALSE;
                                                       END_IF
												END_IF

	JAW_HOMING_STATES.HomeComplete:				MoveToPosition(2, 1000,1000,2583);
												homingState := JAW_HOMING_STATES.MovingToTwoInches;

	JAW_HOMING_STATES.MovingToTwoInches : 		timerHomeDelay.PT := T#200MS;
												timerHomeDelay.IN := TRUE;
												IF timerHomeDelay.Q THEN
													IF (NOT Moving AND InPosition) THEN
														homingState := JAW_HOMING_STATES.SetLimits;
														timerHomeDelay.IN := FALSE;
                                                       END_IF
												END_IF

	JAW_HOMING_STATES.SetLimits :				commandSuccessful := FALSE;
												ExecuteStoredProgram(3);
												homingState := JAW_HOMING_STATES.Idle;

END_CASE

METHOD HomeNow

_homeNow := TRUE;

//{warning 'add method implementation '}
METHOD Stop

commandSuccessful := FALSE;
commands.StopCrash := TRUE;

(* ---- FB_AppliedMotionStepServoMBBase.st ---- *)
FUNCTION_BLOCK FB_AppliedMotionStepServoMBBase IMPLEMENTS IPositionableMotor, IStoredProgramMotor
VAR_INPUT
    modbusInputParameters : ARRAY[0 .. 124] OF WORD;        //This is the input array of words of raw Modbus registers
    stepsPerInchSetpoint : INT;                                        //Steps per inch setpoint
    reversePolarity : BOOL;                                    //0 = Normal, 1 = reversed polarity for display
    pointToPointAccelSetpoint : INT;        //Point-to-Point Acceleration (AC) Setpoint
    pointToPointDecelSetpoint : INT;        //Point-to-Point Deceleration (DE) Setpoint
    velocitySetpoint : INT;                //Velocity (VE) Setpoint
    distanceSetpointInches : REAL;        //Distance setpoint in inches Setpoint
    moveDistanceManualPB : BOOL;            //Move distance pushbutton
    movePositionManualPB : BOOL;            //Move position pushbutton
END_VAR
VAR_IN_OUT
    //slave : IoDrvModbusTCP.ModbusTCPSlave;                    //Slave ModbusTCP Object
END_VAR
VAR
    ModbusLongHandler : ModbusLongHandlerFB();
    absolutePositionSteps : ModbusLongType; //Immediate Absolute Position in steps
    distanceSteps : ModbusLongType;    //Point-to-Point Distance (DI) Input from Drive Combined
    distanceToMoveInSteps : ModbusLongType;        //Distance Setpoint to Drive
    stepServoStatusRaw : INT; //Raw step servo status over modbus
    commandSuccessful : BOOL;    //Modbus Command was successful
    homeRequiredIndication : BOOL; //Home required indication.
    //commandAcked : BOOL;        //Command acked from "send" function blocks
    interfaceToPass : IFault;
    faultListRegisterSuccess : BOOL;        // Registering in fault list successful
    _faulted : BOOL;                    // Motor Faulted
END_VAR
VAR_OUTPUT
    absolutePositonInches : REAL; //Immediate Absolute Positon in inches
    distanceInches : REAL;            //Distance from Drive converted to inches
    homeAccel : INT;    //Home Acceleration (HA) Input from Drive
    homeCurrentLimit : INT;    //Home Hard Stop current limit (HC) Input from Drive
    homeDecel : INT;    //Home Deceleration (HL) Input from Drive
    homeVelocity : INT;    //Home Speed (HV) from Drive
    jogAccel : INT;    //Jog Acceleration (AC) Input from Drive
    jogDecel : INT;    //Jog Deceleration (DE) Input from Drive
    jogVelocity : INT;    //Jog Speed from Drive
    pointToPointAccel : INT;    //Point-to-Point Acceleration (AC) Input from Drive
    pointToPointDecel : INT;    //Point-to-Point Deceleration (DE) Input from Drive
    velocity : INT;    //Velocity (VE) Input from Drive
    status : StepServoStatusFB; //Status of servo
    QSegmentRunning : INT; //Current Q program running from Drive
END_VAR

METHOD Execute
VAR_INPUT
END_VAR

//    Function Block: AppliedMotionStepServo
//    Description: This block provides an abstraction for a Applied Motion Step Servo
//    Created by: Ben Hess
//    Created Date: April 2nd, 2018

//Map raw Modbus Registers to parameters
absolutePositionSteps.highWord := modbusInputParameters[6];
absolutePositionSteps.lowWord := modbusInputParameters[7];
distanceSteps.highWord := modbusInputParameters[30];
distanceSteps.lowWord := modbusInputParameters[31];
jogAccel := WORD_TO_INT(modbusInputParameters[46]);
jogDecel := WORD_TO_INT(modbusInputParameters[47]);
jogVelocity := WORD_TO_INT(modbusInputParameters[48]);
pointToPointAccel := WORD_TO_INT(modbusInputParameters[27]);
pointToPointDecel := WORD_TO_INT(modbusInputParameters[28]);
velocity := WORD_TO_INT(modbusInputParameters[29]);
stepServoStatusRaw := WORD_TO_INT(modbusInputParameters[1]);
QSegmentRunning := WORD_TO_INT(modbusInputParameters[17]);

//Convert Distance setpoint to steps.  Reverse polarity for display purposes if needed.
//oDistanceSteps.displayValue := REAL_TO_DINT((oDistanceInches) * stepsPerInch);
//oDistanceSteps.rawValue := REAL_TO_DINT((oDistanceInches ) * stepsPerInch);
//DistanceSteps.displayValue := DistanceSteps.rawValue;
distanceInches := (DINT_TO_REAL(distanceSteps.displayValue) / INT_TO_REAL(stepsPerInchSetpoint));
absolutePositionSteps.displayValue := absolutePositionSteps.rawValue;
absolutePositonInches := (DINT_TO_REAL(absolutePositionSteps.displayValue) / INT_TO_REAL(stepsPerInchSetpoint));

//Homing required from motor - for now just if there was an initialization seen.
homeRequiredIndication S= status.initializing OR Globals.firstScan;

IF reversePolarity THEN
    //oDistanceSteps.rawValue := oDistanceSteps.rawValue * -1;
    distanceInches := distanceInches * -1;
    absolutePositonInches := absolutePositonInches * -1;
END_IF

//Get Servo Status and unpack
status(statusCode := StepServoStatusRaw);

//Bit-packing for LONG types over Modbus
ModbusLongHandler.Pack(distanceSteps);
ModbusLongHandler.Pack(absolutePositionSteps);

//Manual moves for motor
IF moveDistanceManualPB THEN
    MoveDistance(distance := distanceSetpointInches, acceleration := pointToPointAccelSetpoint, deceleration := pointToPointDecelSetpoint, velocity := velocitySetpoint);
    moveDistanceManualPB := FALSE;
END_IF

IF movePositionManualPB THEN
    MoveToPosition(position := distanceSetpointInches, acceleration := pointToPointAccelSetpoint, deceleration := pointToPointDecelSetpoint, velocity := velocitySetpoint);
    movePositionManualPB := FALSE;
END_IF

{attribute 'monitoring' := 'variable'}
PROPERTY HomeRequired : BOOL

{attribute 'monitoring' := 'variable'}
PROPERTY CommandAcknowledged : BOOL

METHOD ExecuteStoredProgram
VAR_INPUT
    (*Program number to execute*)
    programNumber    : INT;
END_VAR

{attribute 'monitoring' := 'variable'}
PROPERTY Homing : BOOL

{attribute 'monitoring' := 'variable'}
PROPERTY ActiveStoredProgramNumber : INT

{attribute 'monitoring' := 'variable'}
PROPERTY Moving : BOOL

//{warning 'add method implementation '}
METHOD MoveDistance
VAR_INPUT
    (*Distance to move in inches*)
    distance    : REAL;
    (*Acceleration in RPM/sec*)
    acceleration    : INT;
    (*Deceleration in RPM/sec*)
    deceleration    : INT;
    (*Velocity in .25RPM*)
    velocity    : INT;
END_VAR

{attribute 'monitoring' := 'variable'}
PROPERTY InPosition : BOOL

METHOD HomeNow

//{warning 'add method implementation '}
METHOD Stop

{attribute 'monitoring' := 'variable'}
PROPERTY CurrentPosition : REAL  //Current motor position in Inches

//{warning 'add method implementation '}
METHOD MoveToPosition
VAR_INPUT
    (*Position to move to in inches*)
    position    : REAL;
    (*Acceleration in RPM/sec*)
    acceleration    : INT;
    (*Deceleration in RPM/sec*)
    deceleration    : INT;
    (*Velocity in .25RPM*)
    velocity    : INT;
END_VAR

(* ---- FB_AppliedMotionStepServoTCP.st ---- *)
FUNCTION_BLOCK FB_AppliedMotionStepServoTCP EXTENDS FB_AppliedMotionStepServoMBBase IMPLEMENTS IPositionableMotor
VAR_INPUT
END_VAR
VAR_IN_OUT
    slave : IoDrvModbusTCP.ModbusTCPSlave;                    //Slave ModbusTCP Object
END_VAR
VAR_OUTPUT
END_VAR
VAR
    sendMoveCommand : FB_SendMoveCommandAppliedMotionTCP();
    sendOpcodeCommand :  FB_SendOpcodeCommandAppliedMotionTCP();
END_VAR

sendMoveCommand(Slave := slave);
sendOpcodeCommand(Slave := slave);

commandSuccessful S= (sendMoveCommand.xDone OR sendOpcodeCommand.xDone) AND NOT status.inPosition;

METHOD Stop

commandSuccessful := FALSE;
SendOpcodeCommand.opcode := STEP_SERVO_OPCODES.STOP_MOVE_KILL_BUFFER;
SendOpcodeCommand.Execute();

METHOD MoveToPosition
VAR_INPUT
    (*Position to move to in inches*)
    position    : REAL;
    (*Acceleration in RPM/sec*)
    acceleration    : INT;
    (*Deceleration in RPM/sec*)
    deceleration    : INT;
    (*Velocity in .25RPM*)
    velocity    : INT;
END_VAR

//This method preps the data to send to the drive and triggers the send.
//Set distance and unpack to prep data to send to motor
distanceToMoveInSteps.rawValue := REAL_TO_DINT((position) * stepsPerInchSetpoint);
IF reversePolarity THEN
    distanceToMoveInSteps.rawValue := distanceToMoveInSteps.rawValue * -1;
END_IF
commandSuccessful := FALSE;
ModbusLongHandler.Unpack(distanceToMoveInSteps);
sendMoveCommand.acceleration := acceleration;
sendMoveCommand.deceleration := deceleration;
sendMoveCommand.velocity := velocity;
sendMoveCommand.distanceHighWord := distanceToMoveInSteps.highWord;
sendMoveCommand.distanceLowWord := distanceToMoveInSteps.lowWord;
sendMoveCommand.opcode := STEP_SERVO_OPCODES.FEED_TO_POSITION;
sendMoveCommand.Execute();

METHOD ExecuteStoredProgram
VAR_INPUT
    (*Program number to execute*)
    programNumber    : INT;
END_VAR

//Load program into queue by setting it as parameter 1 and send it and the execute queue opcode
commandSuccessful := FALSE;
SendOpcodeCommand.opcode := STEP_SERVO_OPCODES.QUEUE_LOAD_AND_EXECUTE;
SendOpcodeCommand.Parameter1 := INT_TO_WORD(programNumber);
SendOpcodeCommand.Execute();

METHOD MoveDistance
VAR_INPUT
    distance : REAL;        //Distance to move in inches
    acceleration : INT;        //Acceleration in RPM/sec
    deceleration : INT;        //Deceleration in RPM/sec
    velocity : INT;            //Velocity in .25RPM
END_VAR
//This method preps the data to send to the drive and triggers the send.
//Set distance and unpack to prep data to send to motor
distanceToMoveInSteps.rawValue := REAL_TO_DINT((distance) * stepsPerInchSetpoint);
IF reversePolarity THEN
    distanceToMoveInSteps.rawValue := distanceToMoveInSteps.rawValue * -1;
END_IF
commandSuccessful := FALSE;
ModbusLongHandler.Unpack(distanceToMoveInSteps);
sendMoveCommand.acceleration := acceleration;
sendMoveCommand.deceleration := deceleration;
sendMoveCommand.velocity := velocity;
sendMoveCommand.distanceHighWord := distanceToMoveInSteps.highWord;
sendMoveCommand.distanceLowWord := distanceToMoveInSteps.lowWord;
sendMoveCommand.opcode := STEP_SERVO_OPCODES.FEED_TO_LENGTH;
sendMoveCommand.Execute();

METHOD HomeNow

//Load program 1 into queue by setting it as parameter 1 and send it and the execute queue opcode
ExecuteStoredProgram(QX_PROGRAMS.HOME_HARD_STOP);
HomeRequired := FALSE;

(* ---- FB_CollectionHandlerActiveFaults.st ---- *)
FUNCTION_BLOCK FB_CollectionHandlerActiveFaults
VAR_INPUT
END_VAR
VAR
	Collection: ARRAY[0..GlobalObjects.MAX_FAULTS] OF IFault; // object array
	ObjNames   : ARRAY[0..GlobalObjects.MAX_FAULTS] OF STRING;
	_ArrayOver   : BOOL;
	_BadObj      : INT;
	_DupeObj   : INT;
	_OverObj   : INT;
	_TotalObj   : UINT;
END_VAR

VAR_OUTPUT
	faultActive : BOOL;
END_VAR
//	Function Block: FB_CollectionHandlerActiveFaults
//	Description: This collection handler adds and removes active faults to an array
//				 The add and remove methods are called from FB_Fault
//	Created by: Tom Jacobs
//	Created Date: Friday, September 7, 2018

METHOD RemoveObject
VAR_INPUT
	Obj   : IFault;
END_VAR

VAR
	I   : UINT;
	J : UINT;
END_VAR

FOR I:= 0 TO _TotalObj DO
	IF Collection[I] = Obj THEN
		// object pointer matches - get rid of it
		FOR J := I TO _TotalObj DO
			Collection[J] := Collection[J+1];
			ObjNames[J]:= ObjNames[J+1];
		END_FOR
		_TotalObj := _TotalObj - 1;
		IF _TotalObj = 0 THEN
			faultActive := FALSE;
		END_IF
		RETURN;
	END_IF
END_FOR

METHOD AckAll
VAR_INPUT
END_VAR
VAR
	Cast : IFault;
	Fault : IFault;
	J : UINT;
END_VAR
// For each active fault in the array, ack it.
FOR J:= 0 TO _TotalObj - 1 DO
	IF (__QUERYINTERFACE(Collection[J], Cast)) THEN
		Cast.Ack();
	ELSE
		RETURN;
	END_IF
END_FOR

METHOD AddObject
VAR_INPUT
	Obj   : IFault;
END_VAR
VAR
	I   : UINT;
	J : UINT;
END_VAR
// Add the active fault to the array
FOR J:= 0 TO _TotalObj DO
	IF Collection[J] = Obj THEN
		// object pointer matches - it's already in here
		RETURN;
	END_IF
END_FOR

IF _TotalObj < GlobalObjects.MAX_FAULTS THEN
	Collection[_TotalObj]:= Obj;
	ObjNames[_TotalObj]:= Obj.InstanceName;
	_TotalObj:= _TotalObj + 1;
ELSE
	_ArrayOver:= TRUE;
	_OverObj:= _OverObj + 1;
END_IF

faultActive := TRUE;

(* ---- FB_CollectionHandlerAll.st ---- *)
FUNCTION_BLOCK FINAL FB_CollectionHandlerAll
VAR_INPUT
END_VAR
VAR
	Collection: ARRAY[0..GlobalObjects.MAX_OBJECTS] OF IAllObjects; // object array
	ObjNames   : ARRAY[0..GlobalObjects.MAX_OBJECTS] OF STRING;
	_ArrayOver   : BOOL;
	_BadObj      : INT;
	_DupeObj   : INT;
	_OverObj   : INT;
	_TotalObj   : UINT;
END_VAR

METHOD FINAL AddObject
VAR_INPUT
	Obj   : IAllObjects;
END_VAR
VAR
	AnyObject : IAllObjects;
	Fault : IFault;
	Cylinder : ICylinder;
	PositionableMotor : IPositionableMotor;
	Logger : IMachineLogger;
	Loggable : ILoggable;
	Executable : IExecuteAutomatically;
	Initializable : IInitializable;
	J   : UINT;
END_VAR
IF (__QUERYINTERFACE(Obj, AnyObject)) THEN
   // make sure haven't already added this object
   FOR J:= 1 TO _TotalObj DO
      IF Collection[J] = AnyObject THEN
         // object pointer matches - dupe!
         _DupeObj:= _DupeObj + 1;
         RETURN;
      END_IF
   END_FOR

   IF _TotalObj < GlobalObjects.MAX_OBJECTS THEN
      Collection[_TotalObj]:= AnyObject;
      ObjNames[_TotalObj]:= Obj.InstanceName;
	   _TotalObj:= _TotalObj + 1;
   ELSE
      _ArrayOver:= TRUE;
      _OverObj:= _OverObj + 1;
   END_IF
ELSE
   _BadObj:= _BadObj + 1;
END_IF

// Add object to proper collection based on its interfaces
IF (__QUERYINTERFACE(Obj, Fault)) THEN
	GlobalObjects.CollectionOfFaults.AddObject(Fault);
END_IF

// IF (__QUERYINTERFACE(Obj, Cylinder)) THEN
// 	GlobalObjects.CollectionOfCylinders.AddObject(Cylinder);
// END_IF
//
// IF (__QUERYINTERFACE(Obj, PositionableMotor)) THEN
// 	GlobalObjects.CollectionOfPositionableMotors.AddObject(PositionableMotor);
// END_IF

IF (__QUERYINTERFACE(Obj, Logger)) THEN
	GlobalObjects.CollectionOfLogs.AddObject(Logger);
END_IF

IF (__QUERYINTERFACE(Obj, Loggable)) THEN
	GlobalObjects.CollectionOfLoggable.AddObject(Loggable);
END_IF

IF (__QUERYINTERFACE(Obj, Executable)) THEN
	GlobalObjects.CollectionOfExecutable.AddObject(Executable);
END_IF

IF (__QUERYINTERFACE(Obj, Initializable)) THEN
	GlobalObjects.CollectionOfInitialzable.AddObject(Initializable);
END_IF

(* ---- FB_CollectionHandlerExecutable.st ---- *)
FUNCTION_BLOCK FB_CollectionHandlerExecutable
VAR_INPUT
END_VAR
VAR
	Collection: ARRAY[0..GlobalObjects.MAX_EXECUTEABLE] OF IExecuteAutomatically; // object array
	ObjNames   : ARRAY[0..GlobalObjects.MAX_EXECUTEABLE] OF STRING;
	_ArrayOver   : BOOL;
	_BadObj      : INT;
	_DupeObj   : INT;
	_OverObj   : INT;
	_TotalObj   : UINT;
END_VAR
//	Function Block: FB_CollectionHandlerExecutable
//	Description: This collection handler stores executable FB's to an array
//				 and has a method to execute them all on demand
//	Created by: Ben Hess
//	Created Date: Friday, September 7, 2018

METHOD ExecuteAll
VAR_INPUT
END_VAR
VAR
	Cast : IExecuteAutomatically;
	J : UINT;
END_VAR
// For each executable objest in the array, run its "Execute()" method
FOR J:= 0 TO _TotalObj - 1 DO
	IF (__QUERYINTERFACE(Collection[J], Cast)) THEN
		Cast.Execute();
	ELSE
		RETURN;
	END_IF
END_FOR

METHOD AddObject
VAR_INPUT
	Obj   : IExecuteAutomatically;
END_VAR
VAR
	I   : UINT;
	J : UINT;
END_VAR
// Add the active fault to the array
FOR J:= 0 TO _TotalObj DO
	IF Collection[J] = Obj THEN
		// object pointer matches - it's already in here
		RETURN;
	END_IF
END_FOR

IF _TotalObj < GlobalObjects.MAX_EXECUTEABLE THEN
	Collection[_TotalObj]:= Obj;
	ObjNames[_TotalObj]:= Obj.InstanceName;
	_TotalObj:= _TotalObj + 1;
ELSE
	_ArrayOver:= TRUE;
	_OverObj:= _OverObj + 1;
END_IF

(* ---- FB_CollectionHandlerFaults.st ---- *)
FUNCTION_BLOCK FB_CollectionHandlerFaults
VAR_INPUT
END_VAR
VAR
	Collection: ARRAY[0..GlobalObjects.MAX_FAULTS] OF IFault; // object array
	ObjNames   : ARRAY[0..GlobalObjects.MAX_FAULTS] OF STRING;
	_ArrayOver   : BOOL;
	_BadObj      : INT;
	_DupeObj   : INT;
	_OverObj   : INT;
	_TotalObj   : UINT;
END_VAR

METHOD AckAll
VAR_INPUT
END_VAR
VAR
	J : UINT;
END_VAR
FOR J:= 0 TO _TotalObj - 1 DO
	Collection[J].Ack();
END_FOR

METHOD AddObject
VAR_INPUT
	Obj   : IFault;
END_VAR
VAR
	J   : UINT;
END_VAR
FOR J:= 0 TO _TotalObj DO
	IF Collection[J] = Obj THEN
		// object pointer matches - dupe!
		_DupeObj:= _DupeObj + 1;
		RETURN;
	END_IF
END_FOR

IF _TotalObj < GlobalObjects.MAX_FAULTS THEN
	Collection[_TotalObj]:= Obj;
	ObjNames[_TotalObj]:= Obj.InstanceName;
	_TotalObj:= _TotalObj + 1;
ELSE
	_ArrayOver:= TRUE;
	_OverObj:= _OverObj + 1;
END_IF

(* ---- FB_CollectionHandlerInitializable.st ---- *)
FUNCTION_BLOCK FB_CollectionHandlerInitializable
VAR_INPUT

END_VAR
VAR
	Collection: ARRAY[0..GlobalObjects.MAX_LOGGABLE] OF IInitializable; // object array
	ObjNames   : ARRAY[0..GlobalObjects.MAX_LOGGABLE] OF STRING;
	_ArrayOver   : BOOL;
	_BadObj      : INT;
	_DupeObj   : INT;
	_OverObj   : INT;
	_TotalObj   : UINT;
END_VAR
//	Function Block: FB_CollectionHandlerLoggable
//	Description: This collection handler takes in loggable objects and registers them with a logger.  The FirstScan function should trigger the
//				 RegisterAll() method to register all loggable objects with a logger
//	Created by: Ben Hess
//	Created Date: Tuesday, September 11, 2018

METHOD InitializeAll
VAR_INPUT

END_VAR
VAR
	J : UINT;
	Cast : IInitializable;
END_VAR

FOR J:= 0 TO _TotalObj - 1 DO
	IF (__QUERYINTERFACE(Collection[J], Cast)) THEN
		Cast.Initialize();
	ELSE
		RETURN;
	END_IF
END_FOR

METHOD AddObject
VAR_INPUT
	Obj   : IInitializable;
END_VAR
VAR
	J   : UINT;
END_VAR
FOR J:= 0 TO _TotalObj DO
	IF Collection[J] = Obj THEN
		// object pointer matches - dupe!
		_DupeObj:= _DupeObj + 1;
		RETURN;
	END_IF
END_FOR

IF _TotalObj < GlobalObjects.MAX_LOGGABLE THEN
	Collection[_TotalObj]:= Obj;
	ObjNames[_TotalObj]:= Obj.InstanceName;
	_TotalObj:= _TotalObj + 1;
ELSE
	_ArrayOver:= TRUE;
	_OverObj:= _OverObj + 1;
END_IF

(* ---- FB_CollectionHandlerLoggable.st ---- *)
FUNCTION_BLOCK FB_CollectionHandlerLoggable
VAR_INPUT

END_VAR
VAR
	Collection: ARRAY[0..GlobalObjects.MAX_LOGGABLE] OF ILoggable; // object array
	ObjNames   : ARRAY[0..GlobalObjects.MAX_LOGGABLE] OF STRING;
	_ArrayOver   : BOOL;
	_BadObj      : INT;
	_DupeObj   : INT;
	_OverObj   : INT;
	_TotalObj   : UINT;
	_internalLogger : REFERENCE TO IMachineLogger;
END_VAR
//	Function Block: FB_CollectionHandlerLoggable
//	Description: This collection handler takes in loggable objects and registers them with a logger.  The FirstScan function should trigger the
//				 RegisterAll() method to register all loggable objects with a logger
//	Created by: Ben Hess
//	Created Date: Tuesday, September 11, 2018

METHOD RegisterAll
VAR_INPUT
	internalLogger : IMachineLogger;
END_VAR
VAR
	I   : UINT;
	J : UINT;
	cast : ILoggable;
END_VAR

FOR J:= 0 TO _TotalObj - 1 DO
	IF (__QUERYINTERFACE(Collection[J], Cast)) THEN
		cast.RegisterLogger(internalLogger := internalLogger);
	ELSE
		RETURN;
	END_IF
END_FOR

METHOD AddObject
VAR_INPUT
	Obj   : ILoggable;
END_VAR
VAR
	J   : UINT;
END_VAR
FOR J:= 0 TO _TotalObj DO
	IF Collection[J] = Obj THEN
		// object pointer matches - dupe!
		_DupeObj:= _DupeObj + 1;
		RETURN;
	END_IF
END_FOR

IF _TotalObj < GlobalObjects.MAX_LOGGABLE THEN
	Collection[_TotalObj]:= Obj;
	ObjNames[_TotalObj]:= Obj.InstanceName;
	_TotalObj:= _TotalObj + 1;
ELSE
	_ArrayOver:= TRUE;
	_OverObj:= _OverObj + 1;
END_IF

(* ---- FB_CycleCounter.st ---- *)
FUNCTION_BLOCK FB_CycleCounter
VAR_INPUT
	reset : BOOL;
END_VAR
VAR_OUTPUT
END_VAR
VAR PERSISTENT RETAIN
    count : UDINT;
END_VAR

IF reset THEN
	THIS^.Clear();
	reset := FALSE;
END_IF

METHOD Increment
VAR_INPUT
END_VAR

count := count + 1;

METHOD Clear
VAR_INPUT
END_VAR

count := 0;

METHOD SetCount
VAR_INPUT
	countSetting : UDINT;
END_VAR

count := countSetting;

(* ---- FB_Cylinder.st ---- *)
FUNCTION_BLOCK FB_Cylinder IMPLEMENTS ICylinder
VAR_INPUT
    mode : DEVICE_MODES;
END_VAR
VAR_OUTPUT
    extendedStatus : BOOL;
    retractedStatus : BOOL;
    extendOutput : BOOL;
    retractOutput : BOOL;
END_VAR
VAR
END_VAR

METHOD Retract

extendOutput := FALSE;
retractOutput := TRUE;

METHOD Extend

extendOutput := TRUE;
retractOutput := FALSE;

METHOD Execute

//Do nothing

(* ---- FB_CylinderFaults.st ---- *)
FUNCTION_BLOCK FB_CylinderFaults
VAR_INPUT
	enable : BOOL;
	extendCommand : BOOL;
	extendedInput : BOOL;
	retractCommand : BOOL;
	retractedInput : BOOL;
	faultTime : TIME := T#2500ms;
END_VAR
VAR_OUTPUT
	failToExtend : BOOL;
	failToRetract : BOOL;
END_VAR
VAR
	extendFaultTimer : Standard.TON;
	retractFaultTimer : Standard.TON;
END_VAR
VAR_IN_OUT
END_VAR
extendFaultTimer(PT := faultTime, Q => failToExtend);
retractFaultTimer(PT := faultTime, Q => failToRetract);
IF enable THEN
	IF extendCommand THEN
		retractFaultTimer.IN := FALSE;
		extendFaultTimer.IN := NOT extendedInput;
	ELSIF retractCommand THEN
		extendFaultTimer.IN := FALSE;
		retractFaultTimer.IN := NOT retractedInput;
	ELSE
		retractFaultTimer.IN := FALSE;
		extendFaultTimer.IN := FALSE;
	END_IF
ELSE
	retractFaultTimer.IN := FALSE;
	extendFaultTimer.IN := FALSE;
END_IF

(* ---- FB_CylinderLeak.st ---- *)
FUNCTION_BLOCK FB_CylinderLeak EXTENDS FB_PredictiveMaint
VAR_INPUT
	iExtended : BOOL;
	iRetracted : BOOL;
	maximumStrokeTime : REAL;
END_VAR
VAR_OUTPUT
	strokeTime : REAL;
END_VAR
VAR
	strokeTimer : TON := (PT := T#1H);
	extendedONS : R_TRIG;
	retractedONS : R_TRIG;
END_VAR

extendedONS(CLK := iExtended);
retractedONS(CLK := iRetracted);

IF extendedONS.Q OR retractedONS.Q THEN
	strokeTime := TO_REAL(strokeTimer.ET) / 1000;
END_IF

strokeTimer(IN := NOT iExtended AND NOT iRetracted);

(* ---- FB_CylinderWithFeedback.st ---- *)
FUNCTION_BLOCK FB_CylinderWithFeedback EXTENDS FB_Cylinder IMPLEMENTS ICylinder, IFault
VAR_INPUT
    extendedFeedbackInput : BOOL;    //Extended feedback input from I/O
    retractedFeedbackInput : BOOL;    //Retracted feedback input from I/O
    extendFaultDelay : INT := 1000;        //Extend fault delay in MS
    retractFaultDelay : INT := 1000;        //Retract fault delay in MS
    faultMonitoring : BOOL;                    //Fault monitoring enabled if true
END_VAR
VAR_OUTPUT
    failedToExtend : FB_Fault;            //Failed to Extend Fault
    failedToRetract : FB_Fault;            //Failed to Retract Fault
END_VAR
VAR
    faultIndication : BOOL;            //Overall fault status of cylinder
    extendFaultTimer : TON;            //Extend Fault Timer
    retractFaultTimer : TON;        //Retract Fault Timer
    resetFaults : BOOL;                //Reset faults
END_VAR

METHOD Execute

//This code monitors the positon of the cylinder and raises a fault if the cylinder doesn't reach its
//desired postion within the specified time.

//Initialize timers
extendFaultTimer(PT := INT_TO_TIME(extendFaultDelay));
retractFaultTimer(PT := INT_TO_TIME(retractFaultDelay));

//Only enable timers if we are to be monitoring faults
IF faultMonitoring THEN
    extendFaultTimer.IN := (extendOutput AND NOT extendedFeedbackInput);
    retractFaultTimer.IN := (retractOutput AND NOT retractedFeedbackInput);
ELSE
        extendFaultTimer.IN := FALSE;
        retractFaultTimer.IN := FALSE;
END_IF

//Rasie the alarms
failedToExtend.faultTrigger := extendFaultTimer.Q;
failedToRetract.faultTrigger := retractFaultTimer.Q;

//Set overall fault indication
//faultIndication := failedToExtend.Active OR failedToRetract;

(* ---- FB_DriveTemp.st ---- *)
FUNCTION_BLOCK FB_DriveTemp EXTENDS FB_PredictiveMaint
VAR_INPUT
	iDriveTemp : DINT;
	maxTemp : REAL;
END_VAR
VAR_OUTPUT
	DriveTemp : REAL;
END_VAR
VAR
END_VAR

DriveTemp := TO_REAL(iDriveTemp) / 10.0;

(* ---- FB_Fault.st ---- *)
FUNCTION_BLOCK FINAL FB_Fault IMPLEMENTS IFault, ILoggable, IExecuteAutomatically
VAR_INPUT
	ackCommand : BOOL;
	faultTrigger : BOOL;
END_VAR
VAR_OUTPUT
	acknowledged : BOOL;
	active : BOOL;
END_VAR
VAR
	_active : BOOL;
	_acked : BOOL;
	_ackCommand : BOOL;
	_logger : IMachineLogger;
	ackCommandOSR : R_TRIG;
	faultTriggerONS : FB_ONS;
	activeONS : FB_ONS;
	_instanceName : STRING;
END_VAR
VAR_IN_OUT

END_VAR

METHOD Execute

//	Function Block: FB_Fault
//	Description: Faults should be of this FB type.
//  An associated FaultType variable needs to be declared in the HMIData global variable list in order to be exposed via OPCUA
//	Implementation should look as follows:
//
//  *** Instantiate the fault with constructor that contains the fault name: ***
//  VAR (*Faults*)
//		exampleFault1 : FB_Fault(name := CONCAT(_prefix,  'Example Fault 1'));
//		exampleFault2 : FB_Fault(name := CONCAT(_prefix,  'Example Fault 2'));
//  END_VAR
//
//  *** In alarm area of FB call the fault(s). refHMIFaults is passed in from above***
//  IF __ISVALIDREF(refHMIFaults) THEN
//		exampleFault1(HMIFault := refHMIFaults.exampleFault1);
//		exampleFault2(HMIFault := refHMIFaults.exampleFault2, faultTrigger := someFaultCondition);
//  END_IF
//
//	*** Either assign faultTrigger in call (as in exampleFault2 above) or set it later in logic
//	exampleFault1.faultTrigger := someFaultCondition;
//
//	Created by: Ben Hess
//	Created Date: Tuesday, May 22, 2018

{warning 'TODO: Add reference to device faulted indicaiton?'}
ackCommandOSR(CLK := _ackCommand);
faultTriggerONS(CLK := faultTrigger);
activeONS(CLK := _active);

IF faultTriggerONS.OSR THEN
	Trigger();
END_IF

IF ackCommandOSR.Q THEN
	_acked := TRUE;
	_ackCommand := FALSE;
END_IF

IF _acked AND NOT faultTrigger THEN
	_active := FALSE;
	_acked := FALSE;
END_IF

IF activeONS.OSF THEN
	GlobalObjects.CollectionOfActiveFaults.RemoveObject(THIS^);
	_logger.AddLogItem(CONCAT(InstanceName, ' Cleared'));
END_IF

// The following is for external communication to HMI etc.
IF ackCommand THEN
	Ack();
	ackCommand := FALSE;
END_IF
active := _active;
acknowledged := _acked;

PROPERTY InstanceName : STRING

METHOD RegisterLogger
VAR_INPUT
	internalLogger : IMachineLogger;
END_VAR

_logger := internalLogger;

METHOD Ack
IF _ackCommand OR _acked THEN
	RETURN;
END_IF
_acked := TRUE;
// Log the ACK.
_logger.AddLogItem(CONCAT(InstanceName,  ' Acked'));

METHOD Trigger

IF _active = TRUE THEN
	RETURN;
END_IF
_active := TRUE;
GlobalObjects.CollectionOfActiveFaults.AddObject(THIS^);
IF _logger <> 0 THEN
	_logger.AddLogItem(CONCAT(InstanceName,  ' Active'));
END_IF

METHOD FB_Init : BOOL
VAR_INPUT
  bInitRetains : BOOL; // TRUE: the retain variables are initialized (reset warm / reset cold)
  bInCopyCode : BOOL;  // TRUE: the instance will be copied to the copy code afterward (online change)
  name : STRING;
END_VAR

_instanceName := name;
GlobalObjects.CollectionOfAllObjects.AddObject(THIS^);

(* ---- FB_FaultHandler.st ---- *)
FUNCTION_BLOCK FB_FaultHandler
VAR_INPUT
END_VAR
VAR_OUTPUT
END_VAR
VAR
    faultSourceList : ARRAY[0..100] OF IFault;
    sourcesInList : INT;
END_VAR

METHOD registerFaultSource
VAR_INPUT
     faultSource : REFERENCE TO IFault;
END_VAR

faultSourceList[sourcesInList]:= faultSource;
sourcesInList:= sourcesInList + 1;

(* ---- FB_FestoMotor.st ---- *)
FUNCTION_BLOCK FB_FestoMotor IMPLEMENTS IPositionableMotor, IStoredProgramMotor
VAR_INPUT
    deviceType : FML.E_FML_DEVICE_TYPE;                            //Must define drive type
    isFPCActive : BOOL;
    ptrReadFHPPRegister : POINTER TO WORD;
    ptrReadFPCRegister : POINTER TO WORD;
    ptrWriteFHPPRegister : POINTER TO WORD;
    ptrWriteFPCRegister : POINTER TO WORD;                                        //Toggle if FPC(Festo Parameter Chanel) is active or not
END_VAR
VAR_IN_OUT
    //modbusReadRegisters :  ARRAY[0..7] OF WORD;        //Inputs from drive
    //modbusWriteRegisters : ARRAY[0..7] OF WORD;    //Outputs to write to drive

END_VAR
VAR_OUTPUT
END_VAR
VAR
    //Required datatypes for the Festo motor blocks
    FHPP_IN     :ARRAY[0..7] OF BYTE;
    FHPP_OUT     :ARRAY[0..7] OF BYTE;
    FPC_IN         :ARRAY[0..7] OF BYTE;
    FPC_OUT     :ARRAY[0..7] OF BYTE;
    ReadAxis            :FML.FML_Read;
    DATA_REF_Axis         :FML.DT_FML_REF;
    CRTL_Axis            :FML.FHPP_CTRL;
    PNU_Axis            :FML.FPC_PNU;
    MULTI_Axis            :FML.FPC_MULTI;
    DIRMP_Axis            :FML.FPC_DIRMP;
    DIAG_Axis            :FML.FPC_DIAG;
    DIAG_BUFF_Axis        :FML.FPC_DIAG_BUFFER;
    DATA_OBJECT_Axis    :FML.FPC_DATA_OBJECT;
    FILE_Axis            :FML.FPC_FILE;
    FILE_ARRAY_Axis        :FML.FPC_FILE_ARRAY;
    WriteAxis            :FML.FML_Write;

    //Regular variables
    ptrModbusMemory : POINTER TO ARRAY[0..7] OF BYTE;
    commandSuccessful : BOOL;    //Modbus Command was successful
    homeRequiredIndication : BOOL; //Home required indication
    homingActive : BOOL;            //Homing active
    removeStartCommandTimer : Standard.TON := (PT := T#100MS);
    startAckONS : Standard.R_TRIG;
    _sendStart : BOOL;
END_VAR
VAR_STAT
    //Make these static to share amongst all instances of the Festo motors
    ARY_DATA_FILE        :ARRAY[0..25000] OF BYTE;
    MultiParam             :ARRAY [0..7] OF DT_FML_PRM_DESCRIPTION :=[
                                            (PNU:=404, SUBINDEX:=1, ACCESS:=0, VALUE:=0, LENGTH:=0),
                                            (PNU:=404, SUBINDEX:=1, ACCESS:=1, VALUE:=100, LENGTH:=4),
                                            (PNU:=404, SUBINDEX:=1, ACCESS:=0, VALUE:=0, LENGTH:=0),
                                            (PNU:=404, SUBINDEX:=2, ACCESS:=0, VALUE:=0, LENGTH:=0),
                                            (PNU:=404, SUBINDEX:=2, ACCESS:=1, VALUE:=200, LENGTH:=4),
                                            (PNU:=404, SUBINDEX:=2, ACCESS:=0, VALUE:=0, LENGTH:=0),
                                            (PNU:=404, SUBINDEX:=1, ACCESS:=1, VALUE:=111, LENGTH:=4),
                                            (PNU:=404, SUBINDEX:=1, ACCESS:=0, VALUE:=0, LENGTH:=0)];

END_VAR

METHOD ExecuteStoredProgram
VAR_INPUT
    (*Program number to execute*)
    programNumber    : INT;
END_VAR

InitDrive();
IF InPosition AND CRTL_Axis.ActualRecordNo = programNumber THEN
    commandSuccessful := TRUE;
ELSE
    CRTL_Axis.RecordNo := programNumber;
    _sendStart := TRUE;
END_IF

{attribute 'monitoring' := 'variable'}
PROPERTY CommandAcknowledged : BOOL

{attribute 'monitoring' := 'variable'}
PROPERTY CurrentPosition : REAL

PROPERTY Homing : BOOL

{attribute 'monitoring' := 'variable'}
PROPERTY InPosition : BOOL

PROPERTY HomeRequired : BOOL

METHOD Execute
VAR_INPUT
END_VAR

//Check to make sure we have a valid reference.  Disable complier warning since we're doing the check
//{warning disable C0371}
(*
IF NOT __ISVALIDREF(ptrReadFHPPRegister)
    OR NOT __ISVALIDREF(ptrReadFPCRegister)
    OR NOT __ISVALIDREF(ptrWriteFHPPRegister)
    OR NOT __ISVALIDREF(ptrWriteFPCRegister)
THEN
     RETURN;
END_IF
*)

//Convert array of bytes to array of words. Playin' with pointers!
ptrModbusMemory := ptrReadFHPPRegister;
FHPP_IN := ptrModbusMemory^;
ptrModbusMemory := ptrReadFPCRegister;
FPC_IN := ptrModbusMemory^;
ptrModbusMemory := ptrWriteFHPPRegister;
ptrModbusMemory^ := FHPP_OUT;
ptrModbusMemory := ptrWriteFPCRegister;
ptrModbusMemory^ := FPC_OUT;

// Function block calls for axis
ReadAxis(
    FML_REF            := DATA_REF_Axis,
    Modbus            := FALSE,
    HighByteFirst    := TRUE,
    DeviceType        := deviceType,
    FPC_active        := isFPCActive,

    FHPP_Source        := FHPP_IN,
    FPC_Source        := FPC_IN);
CRTL_Axis(
    FML_REF            := DATA_REF_Axis);
PNU_Axis(
    FML_REF            := DATA_REF_Axis);
MULTI_Axis(
    FML_REF            := DATA_REF_Axis,
    SizeOfParam        := SIZEOF(MultiParam),
    AdrOfParam        := ADR(MultiParam));
DIRMP_Axis(
    FML_REF            := DATA_REF_Axis);
DIAG_Axis(
    FML_REF            := DATA_REF_Axis);
DIAG_BUFF_Axis(
    FML_REF            := DATA_REF_Axis);
DATA_OBJECT_Axis(
    FML_REF            := DATA_REF_Axis);
FILE_Axis(
    FML_REF            := DATA_REF_Axis);
FILE_ARRAY_Axis(
    FML_REF            := DATA_REF_Axis,
    SizeOfFileArray    := SIZEOF(ARY_DATA_FILE),
    AdrOfFileArray    := ADR(ARY_DATA_FILE));
WriteAxis(
    FML_REF            := DATA_REF_Axis,
    FHPP_Target        => FHPP_OUT,
    FPC_Target        => FPC_OUT);
{warning 'TODO: Remove this hack to clear start command if error occurs'}
removeStartCommandTimer(IN := CRTL_Axis.StartTask OR CRTL_Axis.AckStart);
//removeStartCommandTimer(IN := CRTL_Axis.AckStart);
startAckONS(CLK := CRTL_Axis.AckStart);
//IF removeStartCommandTimer.Q THEN
IF _sendStart AND NOT CRTL_Axis.AckStart THEN
    CRTL_Axis.StartTask := TRUE;
    _sendStart := FALSE;
END_IF

IF startAckONS.Q OR removeStartCommandTimer.Q THEN
    CRTL_Axis.StartTask := FALSE;
    commandSuccessful := TRUE;
END_IF
//Set Home required indication
homeRequiredIndication S= NOT CRTL_Axis.HomingValid;
//commandSuccessful S= CRTL_Axis.AckStart;
//{warning restore C0371}

{attribute 'monitoring' := 'variable'}
PROPERTY ActiveStoredProgramNumber : INT

METHOD Stop

commandSuccessful := FALSE;
CRTL_Axis.EnableDrive := TRUE;
CRTL_Axis.Halt := TRUE;
CRTL_Axis.Stop := FALSE;

METHOD PRIVATE InitDrive
VAR_INPUT
END_VAR

//Initialize the drive to prepare for a move
CRTL_Axis.EnableDrive := TRUE;
CRTL_Axis.Halt := TRUE;
CRTL_Axis.Stop := TRUE;
//CRTL_Axis.StartTask := FALSE;
commandSuccessful := FALSE;

PROPERTY Moving : BOOL

{warning 'add method implementation '}
METHOD MoveDistance
VAR_INPUT
    (*Distance to move in inches*)
    distance    : REAL;
    (*Acceleration in RPM/sec*)
    acceleration    : INT;
    (*Deceleration in RPM/sec*)
    deceleration    : INT;
    (*Velocity in .25RPM*)
    velocity    : INT;
END_VAR

{warning 'add method implementation '}
METHOD MoveToPosition
VAR_INPUT
    (*Position to move to in inches*)
    position    : REAL;
    (*Acceleration in RPM/sec*)
    acceleration    : INT;
    (*Deceleration in RPM/sec*)
    deceleration    : INT;
    (*Velocity in .25RPM*)
    velocity    : INT;
END_VAR

METHOD HomeNow

CRTL_Axis.StartHoming := TRUE;

(* ---- FB_GetTime.st ---- *)
FUNCTION_BLOCK FB_GetTime
VAR_INPUT
END_VAR
VAR_OUTPUT
    currentDateAndTime : DATE_AND_TIME;

END_VAR
VAR
    iState                    : INT;
    udiUtcTime             : UDINT;
    udiUtcTimeLocal     : UDINT;
    strTimeDate         : SYSTIMEDATE;
    strTimeDateLocal     : SYSTIMEDATE;
    dtDateTimeUTC        : DATE_AND_TIME;
    timeLeftTime        : TIME;
    timeLeftDWORD        : DWORD;
    dDateUTC            : DATE;
    todTimeOfDayUTC        : TOD;

    tSysStartTime        : TIME;
    systimeStartNano    : SYSTIME;
    udiStartTimeResult    : UDINT;

    udiResult             : UDINT;

    GetDateAndTime            : DTU.GetDateAndTime;
    SetTimeZoneInformation    : DTU.SetTimeZoneInformation;

    dtCurrent                : DATE_AND_TIME;
    dtConcated                : DATE_AND_TIME;
    eWeekday                 : RTCLK.WEEKDAY;
    uiYear                     : UINT;
    uiMonth                     : UINT;
    uiDay                     : UINT;
    uiHour                     : UINT;
    uiMinute                 : UINT;
    uiSecond                 : UINT;

    dtuError                : DTU.ERROR;
END_VAR

CASE iState OF

    0:
        iState:= 1;

    1:  // retrieves the target date and time, including the timezone information which was set before
        GetDateAndTime( xExecute:= TRUE);
        IF GetDateAndTime.xDone THEN
            dtCurrent:= GetDateAndTime.dtDateAndTime;
            GetDateAndTime(xExecute:= FALSE);
			currentDateAndTime := dtCurrent;
            //timeLeft := TIME_TO_DT(DT_TO_TIME(targetDate) - DT_TO_TIME(dttarget));
            iState:= 2;
        END_IF
        IF GetDateAndTime.xError THEN
            GetDateAndTime(xExecute:= FALSE);
            iState:= 32767;
        END_IF

    2: (*set a spedific date and time --> returns a variable of type DATE_AND_TIME
         DateConcat --> set only date information --> returns a variable of type DATE
         TODConcat  --> set only the time information  --> returns a variable of TOD (Time of day) *)
        IF dtuError = 0 THEN
            iState := 3;
        ELSE
            iState := 32767;
        END_IF

    3:  (*a DATE_AND_TIME variable is splitted in its parts, like year, month, day etc.
            DateSplit --> the same function for a DATE variable
            TODSplit  --> the same function for a TOD variable *)

        IF dtuError = 0 THEN
            iState:= 1;
        ELSE
            iState:= 32767;
        END_IF

    32767: ; //error

END_CASE

(* ---- FB_HMIFault.st ---- *)
FUNCTION_BLOCK FINAL FB_HMIFault IMPLEMENTS IExecuteAutomatically, IAllObjects, IInitializable
VAR_INPUT
	refFault : REFERENCE TO FB_Fault;
END_VAR
VAR_OUTPUT
END_VAR
VAR
	active : REFERENCE TO BOOL;
	acknowledged : REFERENCE TO BOOL;
	ackCommand : REFERENCE TO BOOL;
	_instanceName : STRING := 'HMI Fault';
END_VAR

PROPERTY InstanceName : STRING

METHOD FB_Init : BOOL
VAR_INPUT
  bInitRetains : BOOL; // TRUE: the retain variables are initialized (reset warm / reset cold)
  bInCopyCode : BOOL;  // TRUE: the instance will be copied to the copy code afterward (online change)
END_VAR

GlobalObjects.CollectionOfAllObjects.AddObject(THIS^);

METHOD FB_Reinit : BOOL
VAR_INPUT
END_VAR

THIS^.Initialize();

METHOD Initialize
VAR_INPUT
END_VAR

active REF= refFault.active;
acknowledged REF= refFault.acknowledged;
ackCommand  REF= refFault.ackCommand;
_instanceName := CONCAT('HMI Fault - ', refFault.InstanceName);

METHOD Execute
VAR

END_VAR

(* ---- FB_HMILight.st ---- *)
FUNCTION_BLOCK FB_HMILight
VAR_INPUT
END_VAR
VAR_OUTPUT
	lightOutput : BOOL;
END_VAR
VAR
	_turnOn : BOOL;
	_blinkFast : BOOL;
	_blinkSlow : BOOL;
	blinker : OSCAT_BASIC.PWM_DC := (F := 1, DC := 0.5);
	slowBlinkSec : REAL := 1;
	fastBlinkSec : REAL := 0.5;
END_VAR

IF _blinkFast THEN
	blinker.F := fastBlinkSec;
ELSIF _blinkSlow THEN
	blinker.F := slowBlinkSec;
END_IF

blinker(F:= , DC:= , Q=> );

lightOutput := _turnOn OR (blinker.Q AND (_blinkFast OR _blinkSlow));

METHOD BlinkSlow
VAR_INPUT
END_VAR

_blinkFast := FALSE;
_blinkSlow := TRUE;
_turnOn := FALSE;

METHOD BlinkFast
VAR_INPUT
END_VAR

_blinkFast := TRUE;
_blinkSlow := FALSE;
_turnOn := FALSE;

METHOD TurnOff
VAR_INPUT
END_VAR

_blinkFast := FALSE;
_blinkSlow := FALSE;
_turnOn := FALSE;

METHOD TurnOn
VAR_INPUT
END_VAR

_blinkFast := FALSE;
_blinkSlow := FALSE;
_turnOn := TRUE;

(* ---- FB_IFMTempSensor.st ---- *)
FUNCTION_BLOCK FB_IFMTempSensor EXTENDS FB_TemperatureSensor
VAR_INPUT
	ptrTemperatureBytes : POINTER TO ARRAY[0..1] OF BYTE;
END_VAR
VAR_OUTPUT
	rtdFailure : FB_Fault(name := 'RTD Failure');
END_VAR
VAR
END_VAR

//	Function Block: FB_IFMTempSensor
//	Description: Implemention of an IFM TP3232 IOLink temperature sensor
//
//	Created by: Ben Hess
//	Created Date: Tuesday, September 11, 2018

METHOD Execute
VAR_INPUT
END_VAR

_rawTemperatureReading := TO_INT(OSCAT_BASIC.WORD_OF_BYTE(B0 := ptrTemperatureBytes^[1], B1 := ptrTemperatureBytes^[0]));
_temperatureReadingC := TO_REAL(_rawTemperatureReading / 10.0);
_temperatureReadingF := OSCAT_BASIC.C_TO_F(_temperatureReadingC);

IF _rawTemperatureReading = 0 AND Globals.machinePowerOK THEN
	rtdFailure.Trigger();
END_IF

(* ---- FB_InternalLogger.st ---- *)
FUNCTION_BLOCK FB_InternalLogger IMPLEMENTS IMachineLogger
VAR_INPUT
END_VAR
VAR_OUTPUT
END_VAR
VAR
	//loggedItems : ARRAY[0..500] OF FaultLogType;
	loggedItems : ARRAY[0..GLobals.MAX_LOGGED_ITEMS] OF LogMessageType;
	numOfLogEntries : UINT;
	logFull : BOOL;
	RTC : FB_GetTime();
	clearLog : BOOL;
	i : UINT;
END_VAR

//	Function Block: FB_Logger
//	Description: This is an internal logger for reference within Codesys.  It is an array that can be displayed on the TargetVisu/WebVisu
//
//	Created by: Ben Hess
//	Created Date: Tuesday, September 11, 2018

RTC();

IF clearLog THEN
	FOR i := 0 TO numOfLogEntries BY 1 DO
		loggedItems[i].logMessage := '';
		loggedItems[i].logTime := DT#1970-1-1-1:0:0;
	END_FOR
	numOfLogEntries := 0;
	logFull := FALSE;
	clearLog := FALSE;
END_IF

PROPERTY InstanceName : STRING

METHOD AddLogItem
VAR_INPUT
	message : STRING;
END_VAR

FOR i := Globals.MAX_LOGGED_ITEMS -1 TO 1 BY -1 DO
		loggedItems[i] := loggedItems[i-1];
END_FOR

loggedItems[0].logMessage := message;
loggedItems[0].logTime := RTC.currentDateAndTime;
